	W =  -167.363 deg,	P =     0.000 deg,	R =  -164.964 deg
};
P[653]{
   GP1:
	UF : 7, UT : 3,	CONFIG : 'F U T, 0, 0, 0',
	X =   -22.566  mm,	Y =   363.777  mm,	Z =     0.000  mm,
	W =  -167.363 deg,	P =     0.000 deg,	R =  -161.468 deg
};
P[654]{
   GP1:
	UF : 7, UT : 3,	CONFIG : 'F U T, 0, 0, 0',
	X =   -44.583  mm,	Y =   361.733  mm,	Z =     0.000  mm,
	W =  -167.363 deg,	P =     0.000 deg,	R =  -157.902 deg
};
P[655]{
   GP1:
	UF : 7, UT : 3,	CONFIG : 'F U T, 0, 0, 0',
	X =   -66.134  mm,	Y =   358.425  mm,	Z =     0.000  mm,
	W =  -167.363 deg,	P =     0.000 deg,	R =  -154.243 deg
};
P[656]{
   GP1:
	UF : 7, UT : 3,	CONFIG : 'F U T, 0, 0, 0',
	X =   -66.134  mm,	Y =   358.425  mm,	Z =     0.000  mm,
	W =  -167.363 deg,	P =     0.000 deg,	R =  -154.243 deg
};
P[657]{
   GP1:
	UF : 7, UT : 3,	CONFIG : 'F U T, 0, 0, 0',
	X =   -66.134  mm,	Y =   358.425  mm,	Z =     0.000  mm,
	W =  -167.363 deg,	P =     0.000 deg,	R =  -154.243 deg
};
P[658]{
   GP1:
	UF : 7, UT : 3,	CONFIG : 'F U T, 0, 0, 0',
	X =   -66.134  mm,	Y =   358.425  mm,	Z =     0.000  mm,
	W =  -167.363 deg,	P =     0.000 deg,	R =  -154.243 deg
};
P[659]{
   GP1:
	UF : 7, UT : 3,	CONFIG : 'F U T, 0, 0, 0',
	X =   -95.933  mm,	Y =   351.637  mm,	Z =     0.000  mm,
	W =  -167.364 deg,	P =     0.000 deg,	R =  -149.101 deg
};
P[660]{
   GP1:
	UF : 7, UT : 3,	CONFIG : 'F U T, 0, 0, 0',
	X =   -95.933  mm,	Y =   351.637  mm,	Z =     0.000  mm,
	W =  -167.364 deg,	P =     0.000 deg,	R =  -149.101 deg
};
P[661]{
   GP1:
	UF : 7, UT : 3,	CONFIG : 'F U T, 0, 0, 0',
	X =   -95.933  mm,	Y =   351.637  mm,	Z =     0.000  mm,
	W =  -167.364 deg,	P =     0.000 deg,	R =  -149.101 deg
};
P[662]{
   GP1:
	UF : 7, UT : 3,	CONFIG : 'F U T, 0, 0, 0',
	X =   -95.933  mm,	Y =   351.637  mm,	Z =     0.000  mm,
	W =  -167.364 deg,	P =     0.000 deg,	R =  -149.101 deg
};
P[663]{
   GP1:
	UF : 7, UT : 3,	CONFIG : 'F U T, 0, 0, 0',
	X =  -119.608  mm,	Y =   344.296  mm,	Z =     0.000  mm,
	W =  -167.362 deg,	P =    -0.003 deg,	R =  -145.749 deg
};
P[664]{
   GP1:
	UF : 7, UT : 3,	CONFIG : 'F U T, 0, 0, 0',
	X =  -139.995  mm,	Y =   336.526  mm,	Z =     0.000  mm,
	W =  -167.361 deg,	P =    -0.006 deg,	R =  -142.395 deg
};
P[665]{
   GP1:
	UF : 7, UT : 3,	CONFIG : 'F U T, 0, 0, 0',
	X =  -159.924  mm,	Y =   327.510  mm,	Z =     0.000  mm,
	W =  -167.360 deg,	P =    -0.009 deg,	R =  -139.007 deg
};
P[666]{
   GP1:
	UF : 7, UT : 3,	CONFIG : 'F U T, 0, 0, 0',
	X =  -178.680  mm,	Y =   317.678  mm,	Z =     0.001  mm,
	W =  -167.360 deg,	P =    -0.012 deg,	R =  -135.533 deg
};
P[667]{
   GP1:
	UF : 7, UT : 3,	CONFIG : 'F U T, 0, 0, 0',
	X =  -197.549  mm,	Y =   306.301  mm,	Z =     0.004  mm,
	W =  -167.359 deg,	P =    -0.015 deg,	R =  -132.167 deg
};
P[668]{
   GP1:
	UF : 7, UT : 3,	CONFIG : 'F U T, 0, 0, 0',
	X =  -215.109  mm,	Y =   294.223  mm,	Z =     0.010  mm,
	W =  -167.360 deg,	P =    -0.018 deg,	R =  -128.729 deg
};
P[669]{
   GP1:
	UF : 7, UT : 3,	CONFIG : 'F U T, 0, 0, 0',
	X =  -232.259  mm,	Y =   280.893  mm,	Z =     0.017  mm,
	W =  -167.360 deg,	P =    -0.021 deg,	R =  -125.331 deg
};
P[670]{
   GP1:
	UF : 7, UT : 3,	CONFIG : 'F U T, 0, 0, 0',
	X =  -244.161  mm,	Y =   270.615  mm,	Z =     0.021  mm,
	W =  -167.377 deg,	P =    -0.005 deg,	R =  -122.858 deg
};
P[671]{
   GP1:
	UF : 7, UT : 3,	CONFIG : 'F U T, 0, 0, 0',
	X =  -255.588  mm,	Y =   259.851  mm,	Z =     0.024  mm,
	W =  -167.392 deg,	P =     0.012 deg,	R =  -120.398 deg
};
P[672]{
   GP1:
	UF : 7, UT : 3,	CONFIG : 'F U T, 0, 0, 0',
	X =  -266.547  mm,	Y =   248.605  mm,	Z =     0.021  mm,
	W =  -167.405 deg,	P =     0.031 deg,	R =  -117.928 deg
};
P[673]{
   GP1:
	UF : 7, UT : 3,	CONFIG : 'F U T, 0, 0, 0',
	X =  -276.051  mm,	Y =   238.002  mm,	Z =     0.016  mm,
	W =  -167.466 deg,	P =     0.019 deg,	R =  -115.748 deg
};
P[674]{
   GP1:
	UF : 7, UT : 3,	CONFIG : 'F U T, 0, 0, 0',
	X =  -284.948  mm,	Y =   227.251  mm,	Z =     0.017  mm,
	W =  -167.526 deg,	P =     0.013 deg,	R =  -113.518 deg
};
P[675]{
   GP1:
	UF : 7, UT : 3,	CONFIG : 'F U T, 0, 0, 0',
	X =  -294.786  mm,	Y =   214.339  mm,	Z =     0.044  mm,
	W =  -167.627 deg,	P =    -0.122 deg,	R =  -110.930 deg
};
P[676]{
   GP1:
	UF : 7, UT : 3,	CONFIG : 'F U T, 0, 0, 0',
	X =  -306.175  mm,	Y =   197.743  mm,	Z =     0.197  mm,
	W =  -167.686 deg,	P =    -0.731 deg,	R =  -107.779 deg
};
P[677]{
   GP1:
	UF : 7, UT : 3,	CONFIG : 'F U T, 0, 0, 0',
	X =  -317.263  mm,	Y =   179.431  mm,	Z =     0.730  mm,
	W =  -167.390 deg,	P =    -2.092 deg,	R =  -104.509 deg
};
P[678]{
   GP1:
	UF : 7, UT : 3,	CONFIG : 'F U T, 0, 0, 0',
	X =  -320.981  mm,	Y =   172.696  mm,	Z =     1.000  mm,
	W =  -167.300 deg,	P =    -1.953 deg,	R =  -103.384 deg
};
P[679]{
   GP1:
	UF : 7, UT : 3,	CONFIG : 'F U T, 0, 0, 0',
	X =  -320.981  mm,	Y =   172.696  mm,	Z =     1.000  mm,
	W =  -167.300 deg,	P =    -1.953 deg,	R =  -103.384 deg
};
P[680]{
   GP1:
	UF : 7, UT : 3,	CONFIG : 'F U T, 0, 0, 0',
	X =  -320.981  mm,	Y =   172.696  mm,	Z =     1.000  mm,
	W =  -167.300 deg,	P =    -1.953 deg,	R =  -103.384 deg
};
P[681]{
   GP1:
	UF : 7, UT : 3,	CONFIG : 'F U T, 0, 0, 0',
	X =  -320.981  mm,	Y =   172.696  mm,	Z =     1.000  mm,
	W =  -167.300 deg,	P =    -1.953 deg,	R =  -103.384 deg
};
P[682]{
   GP1:
	UF : 7, UT : 3,	CONFIG : 'F U T, 0, 0, 0',
	X =  -335.149  mm,	Y =   143.280  mm,	Z =     1.000  mm,
	W =  -166.771 deg,	P =     0.958 deg,	R =   -98.400 deg
};
P[683]{
   GP1:
	UF : 7, UT : 3,	CONFIG : 'F U T, 0, 0, 0',
	X =  -335.149  mm,	Y =   143.280  mm,	Z =     1.000  mm,
	W =  -166.771 deg,	P =     0.958 deg,	R =   -98.400 deg
};
P[684]{
   GP1:
	UF : 7, UT : 3,	CONFIG : 'F U T, 0, 0, 0',
	X =  -335.149  mm,	Y =   143.280  mm,	Z =     1.000  mm,
	W =  -166.771 deg,	P =     0.958 deg,	R =   -98.400 deg
};
P[685]{
   GP1:
	UF : 7, UT : 3,	CONFIG : 'F U T, 0, 0, 0',
	X =  -335.149  mm,	Y =   143.280  mm,	Z =     1.000  mm,
	W =  -166.771 deg,	P =     0.958 deg,	R =   -98.400 deg
};
P[686]{
   GP1:
	UF : 7, UT : 3,	CONFIG : 'F U T, 0, 0, 0',
	X =  -339.748  mm,	Y =   131.983  mm,	Z =     0.730  mm,
	W =  -166.786 deg,	P =     1.412 deg,	R =   -96.034 deg
};
P[687]{
   GP1:
	UF : 7, UT : 3,	CONFIG : 'F U T, 0, 0, 0',
	X =  -342.818  mm,	Y =   123.768  mm,	Z =     0.476  mm,
	W =  -167.136 deg,	P =     1.640 deg,	R =   -94.686 deg
};
P[688]{
   GP1:
	UF : 7, UT : 3,	CONFIG : 'F U T, 0, 0, 0',
	X =  -346.796  mm,	Y =   112.170  mm,	Z =     0.189  mm,
	W =  -167.517 deg,	P =     1.060 deg,	R =   -92.897 deg
};
P[689]{
   GP1:
	UF : 7, UT : 3,	CONFIG : 'F U T, 0, 0, 0',
	X =  -351.269  mm,	Y =    97.241  mm,	Z =     0.036  mm,
	W =  -167.527 deg,	P =     0.274 deg,	R =   -90.479 deg
};
P[690]{
   GP1:
	UF : 7, UT : 3,	CONFIG : 'F U T, 0, 0, 0',
	X =  -353.700  mm,	Y =    88.024  mm,	Z =     0.014  mm,
	W =  -167.478 deg,	P =     0.102 deg,	R =   -88.932 deg
};
P[691]{
   GP1:
	UF : 7, UT : 3,	CONFIG : 'F U T, 0, 0, 0',
	X =  -357.903  mm,	Y =    68.887  mm,	Z =     0.006  mm,
	W =  -167.405 deg,	P =     0.015 deg,	R =   -85.835 deg
};
P[692]{
   GP1:
	UF : 7, UT : 3,	CONFIG : 'F U T, 0, 1, 0',
	X =  -361.390  mm,	Y =    47.355  mm,	Z =     0.005  mm,
	W =  -167.391 deg,	P =     0.015 deg,	R =   -82.373 deg
};
P[693]{
   GP1:
	UF : 7, UT : 3,	CONFIG : 'F U T, 0, 1, 0',
	X =  -363.599  mm,	Y =    25.365  mm,	Z =     0.004  mm,
	W =  -167.377 deg,	P =     0.013 deg,	R =   -78.969 deg
};
P[694]{
   GP1:
	UF : 7, UT : 3,	CONFIG : 'F U T, 0, 1, 0',
	X =  -364.492  mm,	Y =     0.000  mm,	Z =     0.000  mm,
	W =  -167.361 deg,	P =     0.009 deg,	R =   -75.580 deg
};
P[695]{
   GP1:
	UF : 7, UT : 3,	CONFIG : 'F U T, 0, 1, 0',
	X =  -364.492  mm,	Y =     0.000  mm,	Z =     0.000  mm,
	W =  -167.361 deg,	P =     0.009 deg,	R =   -75.580 deg
};
P[696]{
   GP1:
	UF : 7, UT : 3,	CONFIG : 'F U T, 0, 1, 0',
	X =  -364.492  mm,	Y =     0.000  mm,	Z =     0.000  mm,
	W =  -167.361 deg,	P =     0.009 deg,	R =   -75.580 deg
};
P[697]{
   GP1:
	UF : 7, UT : 3,	CONFIG : 'F U T, 0, 1, 0',
	X =  -364.492  mm,	Y =     0.000  mm,	Z =     0.000  mm,
	W =  -167.361 deg,	P =     0.009 deg,	R =   -75.580 deg
};
P[698]{
   GP1:
	UF : 7, UT : 3,	CONFIG : 'F U T, 0, 1, 0',
	X =  -361.358  mm,	Y =     0.000  mm,	Z =     0.000  mm,
	W =  -167.361 deg,	P =     0.009 deg,	R =   -75.580 deg
};
P[699]{
   GP1:
	UF : 7, UT : 3,	CONFIG : 'F U T, 0, 1, 0',
	X =  -361.358  mm,	Y =     0.000  mm,	Z =     0.000  mm,
	W =  -167.361 deg,	P =     0.009 deg,	R =   -75.580 deg
};
P[700]{
   GP1:
	UF : 7, UT : 3,	CONFIG : 'F U T, 0, 1, 0',
	X =  -361.358  mm,	Y =     0.000  mm,	Z =     0.000  mm,
	W =  -167.361 deg,	P =     0.009 deg,	R =   -75.580 deg
};
P[701]{
   GP1:
	UF : 7, UT : 3,	CONFIG : 'F U T, 0, 1, 0',
	X =  -361.358  mm,	Y =     0.000  mm,	Z =     0.000  mm,
	W =  -167.361 deg,	P =     0.009 deg,	R =   -75.580 deg
};
P[702]{
   GP1:
	UF : 7, UT : 3,	CONFIG : 'F U T, 0, 1, 0',
	X =  -360.448  mm,	Y =    25.448  mm,	Z =     0.004  mm,
	W =  -167.380 deg,	P =     0.011 deg,	R =   -79.034 deg
};
P[703]{
   GP1:
	UF : 7, UT : 3,	CONFIG : 'F U T, 0, 1, 0',
	X =  -358.205  mm,	Y =    47.576  mm,	Z =     0.004  mm,
	W =  -167.396 deg,	P =     0.011 deg,	R =   -82.501 deg
};
P[704]{
   GP1:
	UF : 7, UT : 3,	CONFIG : 'F U T, 0, 0, 0',
	X =  -354.557  mm,	Y =    69.691  mm,	Z =     0.003  mm,
	W =  -167.412 deg,	P =     0.009 deg,	R =   -85.970 deg
};
P[705]{
   GP1:
	UF : 7, UT : 3,	CONFIG : 'F U T, 0, 0, 0',
	X =  -350.424  mm,	Y =    88.210  mm,	Z =     0.008  mm,
	W =  -167.495 deg,	P =     0.092 deg,	R =   -89.113 deg
};
P[706]{
   GP1:
	UF : 7, UT : 3,	CONFIG : 'F U T, 0, 0, 0',
	X =  -347.970  mm,	Y =    97.380  mm,	Z =     0.026  mm,
	W =  -167.558 deg,	P =     0.268 deg,	R =   -90.637 deg
};
P[707]{
   GP1:
	UF : 7, UT : 3,	CONFIG : 'F U T, 0, 0, 0',
	X =  -343.655  mm,	Y =   111.666  mm,	Z =     0.171  mm,
	W =  -167.608 deg,	P =     1.108 deg,	R =   -93.006 deg
};
P[708]{
   GP1:
	UF : 7, UT : 3,	CONFIG : 'F U T, 0, 0, 0',
	X =  -339.758  mm,	Y =   123.026  mm,	Z =     0.470  mm,
	W =  -167.282 deg,	P =     1.809 deg,	R =   -94.807 deg
};
P[709]{
   GP1:
	UF : 7, UT : 3,	CONFIG : 'F U T, 0, 0, 0',
	X =  -338.361  mm,	Y =   126.823  mm,	Z =     0.600  mm,
	W =  -167.129 deg,	P =     1.834 deg,	R =   -95.529 deg
};
P[710]{
   GP1:
	UF : 7, UT : 3,	CONFIG : 'F U T, 0, 0, 0',
	X =  -334.723  mm,	Y =   136.137  mm,	Z =     0.881  mm,
	W =  -166.917 deg,	P =     1.263 deg,	R =   -97.107 deg
};
P[711]{
   GP1:
	UF : 7, UT : 3,	CONFIG : 'F U T, 0, 0, 0',
	X =  -332.516  mm,	Y =   141.472  mm,	Z =     1.000  mm,
	W =  -166.975 deg,	P =     1.005 deg,	R =   -98.012 deg
};
P[712]{
   GP1:
	UF : 7, UT : 3,	CONFIG : 'F U T, 0, 0, 0',
	X =  -332.516  mm,	Y =   141.472  mm,	Z =     1.000  mm,
	W =  -166.975 deg,	P =     1.005 deg,	R =   -98.012 deg
};
P[713]{
   GP1:
	UF : 7, UT : 3,	CONFIG : 'F U T, 0, 0, 0',
	X =  -332.516  mm,	Y =   141.472  mm,	Z =     1.000  mm,
	W =  -166.975 deg,	P =     1.005 deg,	R =   -98.012 deg
};
P[714]{
   GP1:
	UF : 7, UT : 3,	CONFIG : 'F U T, 0, 0, 0',
	X =  -332.516  mm,	Y =   141.472  mm,	Z =     1.000  mm,
	W =  -166.975 deg,	P =     1.005 deg,	R =   -98.012 deg
};
P[715]{
   GP1:
	UF : 7, UT : 3,	CONFIG : 'F U T, 0, 0, 0',
	X =  -317.920  mm,	Y =   171.762  mm,	Z =     1.000  mm,
	W =  -167.665 deg,	P =    -1.869 deg,	R =  -103.241 deg
};
P[716]{
   GP1:
	UF : 7, UT : 3,	CONFIG : 'F U T, 0, 0, 0',
	X =  -317.920  mm,	Y =   171.762  mm,	Z =     1.000  mm,
	W =  -167.665 deg,	P =    -1.869 deg,	R =  -103.241 deg
};
P[717]{
   GP1:
	UF : 7, UT : 3,	CONFIG : 'F U T, 0, 0, 0',
	X =  -317.920  mm,	Y =   171.762  mm,	Z =     1.000  mm,
	W =  -167.665 deg,	P =    -1.869 deg,	R =  -103.241 deg
};
P[718]{
   GP1:
	UF : 7, UT : 3,	CONFIG : 'F U T, 0, 0, 0',
	X =  -317.920  mm,	Y =   171.762  mm,	Z =     1.000  mm,
	W =  -167.665 deg,	P =    -1.869 deg,	R =  -103.241 deg
};
P[719]{
   GP1:
	UF : 7, UT : 3,	CONFIG : 'F U T, 0, 0, 0',
	X =  -314.044  mm,	Y =   178.741  mm,	Z =     0.714  mm,
	W =  -167.669 deg,	P =    -2.067 deg,	R =  -104.626 deg
};
P[720]{
   GP1:
	UF : 7, UT : 3,	CONFIG : 'F U T, 0, 0, 0',
	X =  -302.748  mm,	Y =   197.275  mm,	Z =     0.167  mm,
	W =  -167.795 deg,	P =    -0.680 deg,	R =  -108.071 deg
};
P[721]{
   GP1:
	UF : 7, UT : 3,	CONFIG : 'F U T, 0, 0, 0',
	X =  -291.275  mm,	Y =   213.833  mm,	Z =     0.025  mm,
	W =  -167.665 deg,	P =    -0.076 deg,	R =  -111.198 deg
};
P[722]{
   GP1:
	UF : 7, UT : 3,	CONFIG : 'F U T, 0, 0, 0',
	X =  -281.263  mm,	Y =   226.842  mm,	Z =     0.007  mm,
	W =  -167.540 deg,	P =     0.044 deg,	R =  -113.765 deg
};
P[723]{
   GP1:
	UF : 7, UT : 3,	CONFIG : 'F U T, 0, 0, 0',
	X =  -272.132  mm,	Y =   237.716  mm,	Z =     0.011  mm,
	W =  -167.474 deg,	P =     0.039 deg,	R =  -116.104 deg
};
P[724]{
   GP1:
	UF : 7, UT : 3,	CONFIG : 'F U T, 0, 0, 0',
	X =  -262.538  mm,	Y =   248.276  mm,	Z =     0.019  mm,
	W =  -167.408 deg,	P =     0.039 deg,	R =  -118.442 deg
};
P[725]{
   GP1:
	UF : 7, UT : 3,	CONFIG : 'F U T, 0, 0, 0',
	X =  -251.581  mm,	Y =   259.374  mm,	Z =     0.023  mm,
	W =  -167.395 deg,	P =     0.018 deg,	R =  -120.883 deg
};
P[726]{
   GP1:
	UF : 7, UT : 3,	CONFIG : 'F U T, 0, 0, 0',
	X =  -240.221  mm,	Y =   269.932  mm,	Z =     0.021  mm,
	W =  -167.380 deg,	P =    -0.002 deg,	R =  -123.334 deg
};
P[727]{
   GP1:
	UF : 7, UT : 3,	CONFIG : 'F U T, 0, 0, 0',
	X =  -228.302  mm,	Y =   280.085  mm,	Z =     0.016  mm,
	W =  -167.364 deg,	P =    -0.020 deg,	R =  -125.793 deg
};
P[728]{
   GP1:
	UF : 7, UT : 3,	CONFIG : 'F U T, 0, 0, 0',
	X =  -211.297  mm,	Y =   293.128  mm,	Z =     0.009  mm,
	W =  -167.363 deg,	P =    -0.018 deg,	R =  -129.084 deg
};
P[729]{
   GP1:
	UF : 7, UT : 3,	CONFIG : 'F U T, 0, 0, 0',
	X =  -194.292  mm,	Y =   304.657  mm,	Z =     0.004  mm,
	W =  -167.362 deg,	P =    -0.015 deg,	R =  -132.493 deg
};
P[730]{
   GP1:
	UF : 7, UT : 3,	CONFIG : 'F U T, 0, 0, 0',
	X =  -176.033  mm,	Y =   315.568  mm,	Z =     0.001  mm,
	W =  -167.362 deg,	P =    -0.012 deg,	R =  -135.789 deg
};
P[731]{
   GP1:
	UF : 7, UT : 3,	CONFIG : 'F U T, 0, 0, 0',
	X =  -157.288  mm,	Y =   325.309  mm,	Z =     0.000  mm,
	W =  -167.362 deg,	P =    -0.009 deg,	R =  -139.100 deg
};
P[732]{
   GP1:
	UF : 7, UT : 3,	CONFIG : 'F U T, 0, 0, 0',
	X =  -138.454  mm,	Y =   333.763  mm,	Z =     0.000  mm,
	W =  -167.362 deg,	P =    -0.006 deg,	R =  -142.478 deg
};
P[733]{
   GP1:
	UF : 7, UT : 3,	CONFIG : 'F U T, 0, 0, 0',
	X =  -118.401  mm,	Y =   341.400  mm,	Z =     0.000  mm,
	W =  -167.363 deg,	P =    -0.003 deg,	R =  -145.771 deg
};
P[734]{
   GP1:
	UF : 7, UT : 3,	CONFIG : 'F U T, 0, 0, 0',
	X =   -95.742  mm,	Y =   348.434  mm,	Z =     0.000  mm,
	W =  -167.364 deg,	P =     0.000 deg,	R =  -149.103 deg
};
P[735]{
   GP1:
	UF : 7, UT : 3,	CONFIG : 'F U T, 0, 0, 0',
	X =   -95.742  mm,	Y =   348.434  mm,	Z =     0.000  mm,
	W =  -167.364 deg,	P =     0.000 deg,	R =  -149.103 deg
};
P[736]{
   GP1:
	UF : 7, UT : 3,	CONFIG : 'F U T, 0, 0, 0',
	X =   -95.742  mm,	Y =   348.434  mm,	Z =     0.000  mm,
	W =  -167.364 deg,	P =     0.000 deg,	R =  -149.103 deg
};
P[737]{
   GP1:
	UF : 7, UT : 3,	CONFIG : 'F U T, 0, 0, 0',
	X =   -95.742  mm,	Y =   348.434  mm,	Z =     0.000  mm,
	W =  -167.364 deg,	P =     0.000 deg,	R =  -149.103 deg
};
P[738]{
   GP1:
	UF : 7, UT : 3,	CONFIG : 'F U T, 0, 0, 0',
	X =   -64.916  mm,	Y =   355.467  mm,	Z =     0.000  mm,
	W =  -167.363 deg,	P =     0.000 deg,	R =  -154.628 deg
};
P[739]{
   GP1:
	UF : 7, UT : 3,	CONFIG : 'F U T, 0, 0, 0',
	X =   -64.916  mm,	Y =   355.467  mm,	Z =     0.000  mm,
	W =  -167.363 deg,	P =     0.000 deg,	R =  -154.628 deg
};
P[740]{
   GP1:
	UF : 7, UT : 3,	CONFIG : 'F U T, 0, 0, 0',
	X =   -64.916  mm,	Y =   355.467  mm,	Z =     0.000  mm,
	W =  -167.363 deg,	P =     0.000 deg,	R =  -154.628 deg
};
P[741]{
   GP1:
	UF : 7, UT : 3,	CONFIG : 'F U T, 0, 0, 0',
	X =   -64.916  mm,	Y =   355.467  mm,	Z =     0.000  mm,
	W =  -167.363 deg,	P =     0.000 deg,	R =  -154.628 deg
};
P[742]{
   GP1:
	UF : 7, UT : 3,	CONFIG : 'F U T, 0, 0, 0',
	X =   -43.097  mm,	Y =   358.757  mm,	Z =     0.000  mm,
	W =  -167.363 deg,	P =     0.000 deg,	R =  -158.018 deg
};
P[743]{
   GP1:
	UF : 7, UT : 3,	CONFIG : 'F U T, 0, 0, 0',
	X =   -21.980  mm,	Y =   360.671  mm,	Z =     0.000  mm,
	W =  -167.363 deg,	P =     0.000 deg,	R =  -161.549 deg
};
P[744]{
   GP1:
	UF : 7, UT : 3,	CONFIG : 'F U T, 0, 0, 0',
	X =     0.061  mm,	Y =   361.358  mm,	Z =     0.000  mm,
	W =  -167.363 deg,	P =     0.000 deg,	R =  -164.959 deg
};
P[745]{
   GP1:
	UF : 7, UT : 3,	CONFIG : 'F U T, 0, 0, 0',
	X =    22.208  mm,	Y =   360.659  mm,	Z =     0.000  mm,
	W =  -167.363 deg,	P =     0.000 deg,	R =  -168.353 deg
};
P[746]{
   GP1:
	UF : 7, UT : 3,	CONFIG : 'F U T, 0, 0, 0',
	X =    43.255  mm,	Y =   358.738  mm,	Z =     0.000  mm,
	W =  -167.363 deg,	P =     0.000 deg,	R =  -171.883 deg
};
P[747]{
   GP1:
	UF : 7, UT : 3,	CONFIG : 'F U T, 0, 0, 0',
	X =    64.916  mm,	Y =   355.467  mm,	Z =     0.000  mm,
	W =  -167.363 deg,	P =     0.000 deg,	R =  -175.272 deg
};
P[748]{
   GP1:
	UF : 7, UT : 3,	CONFIG : 'F U T, 0, 0, 0',
	X =    64.916  mm,	Y =   355.467  mm,	Z =     0.000  mm,
	W =  -167.363 deg,	P =     0.000 deg,	R =  -175.272 deg
};
P[749]{
   GP1:
	UF : 7, UT : 3,	CONFIG : 'F U T, 0, 0, 0',
	X =    64.916  mm,	Y =   355.467  mm,	Z =     0.000  mm,
	W =  -167.363 deg,	P =     0.000 deg,	R =  -175.272 deg
};
P[750]{
   GP1:
	UF : 7, UT : 3,	CONFIG : 'F U T, 0, 0, 0',
	X =    64.916  mm,	Y =   355.467  mm,	Z =     0.000  mm,
	W =  -167.363 deg,	P =     0.000 deg,	R =  -175.272 deg
};
P[751]{
   GP1:
	UF : 7, UT : 3,	CONFIG : 'F U T, 0, 0, 0',
	X =    95.742  mm,	Y =   348.434  mm,	Z =     0.000  mm,
	W =  -167.363 deg,	P =     0.000 deg,	R =   179.209 deg
};
P[752]{
   GP1:
	UF : 7, UT : 3,	CONFIG : 'F U T, 0, 0, 0',
	X =    95.742  mm,	Y =   348.434  mm,	Z =     0.000  mm,
	W =  -167.363 deg,	P =     0.000 deg,	R =   179.209 deg
};
P[753]{
   GP1:
	UF : 7, UT : 3,	CONFIG : 'F U T, 0, 0, 0',
	X =    95.742  mm,	Y =   348.434  mm,	Z =     0.000  mm,
	W =  -167.363 deg,	P =     0.000 deg,	R =   179.209 deg
};
P[754]{
   GP1:
	UF : 7, UT : 3,	CONFIG : 'F U T, 0, 0, 0',
	X =    95.742  mm,	Y =   348.434  mm,	Z =     0.000  mm,
	W =  -167.363 deg,	P =     0.000 deg,	R =   179.209 deg
};
P[755]{
   GP1:
	UF : 7, UT : 3,	CONFIG : 'F U T, 0, 0, 0',
	X =   121.471  mm,	Y =   340.308  mm,	Z =     0.000  mm,
	W =  -167.363 deg,	P =     0.000 deg,	R =   175.407 deg
};
P[756]{
   GP1:
	UF : 7, UT : 3,	CONFIG : 'F U T, 0, 0, 0',
	X =   143.916  mm,	Y =   331.439  mm,	Z =     0.000  mm,
	W =  -167.364 deg,	P =     0.000 deg,	R =   171.611 deg
};
P[757]{
   GP1:
	UF : 7, UT : 3,	CONFIG : 'F U T, 0, 0, 0',
	X =   165.675  mm,	Y =   321.118  mm,	Z =     0.000  mm,
	W =  -167.364 deg,	P =     0.000 deg,	R =   167.801 deg
};
P[758]{
   GP1:
	UF : 7, UT : 3,	CONFIG : 'F U T, 0, 0, 0',
	X =   186.459  mm,	Y =   309.511  mm,	Z =     0.000  mm,
	W =  -167.364 deg,	P =     0.000 deg,	R =   163.968 deg
};
P[759]{
   GP1:
	UF : 7, UT : 3,	CONFIG : 'F U T, 0, 0, 0',
	X =   206.624  mm,	Y =   296.430  mm,	Z =     0.000  mm,
	W =  -167.364 deg,	P =     0.000 deg,	R =   160.166 deg
};
P[760]{
   GP1:
	UF : 7, UT : 3,	CONFIG : 'F U T, 0, 0, 0',
	X =   225.736  mm,	Y =   282.147  mm,	Z =     0.000  mm,
	W =  -167.364 deg,	P =     0.000 deg,	R =   156.350 deg
};
P[761]{
   GP1:
	UF : 7, UT : 3,	CONFIG : 'F U T, 0, 0, 0',
	X =   244.345  mm,	Y =   266.195  mm,	Z =     0.000  mm,
	W =  -167.364 deg,	P =     0.000 deg,	R =   152.581 deg
};
P[762]{
   GP1:
	UF : 7, UT : 3,	CONFIG : 'F U T, 0, 0, 0',
	X =   261.258  mm,	Y =   249.618  mm,	Z =     0.000  mm,
	W =  -167.364 deg,	P =     0.000 deg,	R =   148.718 deg
};
P[763]{
   GP1:
	UF : 7, UT : 3,	CONFIG : 'F U T, 0, 0, 0',
	X =   277.507  mm,	Y =   231.417  mm,	Z =     0.000  mm,
	W =  -167.364 deg,	P =     0.000 deg,	R =   144.979 deg
};
P[764]{
   GP1:
	UF : 7, UT : 3,	CONFIG : 'F U T, 0, 0, 0',
	X =   292.091  mm,	Y =   212.720  mm,	Z =     0.000  mm,
	W =  -167.364 deg,	P =     0.000 deg,	R =   141.122 deg
};
P[765]{
   GP1:
	UF : 7, UT : 3,	CONFIG : 'F U T, 0, 0, 0',
	X =   305.767  mm,	Y =   192.539  mm,	Z =     0.000  mm,
	W =  -167.364 deg,	P =     0.000 deg,	R =   137.342 deg
};
P[766]{
   GP1:
	UF : 7, UT : 3,	CONFIG : 'F U T, 0, 0, 0',
	X =   318.385  mm,	Y =   170.874  mm,	Z =     0.000  mm,
	W =  -167.364 deg,	P =     0.000 deg,	R =   133.523 deg
};
P[767]{
   GP1:
	UF : 7, UT : 3,	CONFIG : 'F U T, 0, 0, 0',
	X =   318.385  mm,	Y =   170.874  mm,	Z =     0.000  mm,
	W =  -167.364 deg,	P =     0.000 deg,	R =   133.523 deg
};
P[768]{
   GP1:
	UF : 7, UT : 3,	CONFIG : 'F U T, 0, 0, 0',
	X =   318.385  mm,	Y =   170.874  mm,	Z =     0.000  mm,
	W =  -167.364 deg,	P =     0.000 deg,	R =   133.523 deg
};
P[769]{
   GP1:
	UF : 7, UT : 3,	CONFIG : 'F U T, 0, 0, 0',
	X =   318.385  mm,	Y =   170.874  mm,	Z =     0.000  mm,
	W =  -167.364 deg,	P =     0.000 deg,	R =   133.523 deg
};
P[770]{
   GP1:
	UF : 7, UT : 3,	CONFIG : 'F U T, 0, 0, 0',
	X =   332.104  mm,	Y =   142.381  mm,	Z =     0.000  mm,
	W =  -167.363 deg,	P =     0.001 deg,	R =   128.768 deg
};
P[771]{
   GP1:
	UF : 7, UT : 3,	CONFIG : 'F U T, 0, 0, 0',
	X =   332.104  mm,	Y =   142.381  mm,	Z =     0.000  mm,
	W =  -167.363 deg,	P =     0.001 deg,	R =   128.768 deg
};
P[772]{
   GP1:
	UF : 7, UT : 3,	CONFIG : 'F U T, 0, 0, 0',
	X =   332.104  mm,	Y =   142.381  mm,	Z =     0.000  mm,
	W =  -167.363 deg,	P =     0.001 deg,	R =   128.768 deg
};
P[773]{
   GP1:
	UF : 7, UT : 3,	CONFIG : 'F U T, 0, 0, 0',
	X =   332.104  mm,	Y =   142.381  mm,	Z =     0.000  mm,
	W =  -167.363 deg,	P =     0.001 deg,	R =   128.768 deg
};
P[774]{
   GP1:
	UF : 7, UT : 3,	CONFIG : 'F U T, 0, 0, 0',
	X =   340.331  mm,	Y =   121.401  mm,	Z =     0.000  mm,
	W =  -167.363 deg,	P =     0.000 deg,	R =   124.654 deg
};
P[775]{
   GP1:
	UF : 7, UT : 3,	CONFIG : 'F U T, 0, 0, 0',
	X =   347.718  mm,	Y =    98.269  mm,	Z =     0.000  mm,
	W =  -167.364 deg,	P =     0.000 deg,	R =   120.888 deg
};
P[776]{
   GP1:
	UF : 7, UT : 3,	CONFIG : 'F U T, 0, 0, 0',
	X =   353.411  mm,	Y =    75.263  mm,	Z =     0.000  mm,
	W =  -167.364 deg,	P =     0.000 deg,	R =   117.027 deg
};
P[777]{
   GP1:
	UF : 7, UT : 3,	CONFIG : 'F U T, 0, 0, 0',
	X =   357.697  mm,	Y =    51.157  mm,	Z =     0.000  mm,
	W =  -167.364 deg,	P =     0.000 deg,	R =   113.281 deg
};
P[778]{
   GP1:
	UF : 7, UT : 3,	CONFIG : 'F U T, 0, 0, 0',
	X =   360.272  mm,	Y =    27.720  mm,	Z =     0.000  mm,
	W =  -167.364 deg,	P =     0.000 deg,	R =   109.419 deg
};
P[779]{
   GP1:
	UF : 7, UT : 3,	CONFIG : 'F U T, 0, 0, 0',
	X =   361.358  mm,	Y =     0.000  mm,	Z =     0.000  mm,
	W =  -167.364 deg,	P =    -0.001 deg,	R =   105.687 deg
};
P[780]{
   GP1:
	UF : 7, UT : 3,	CONFIG : 'F U T, 0, 0, 0',
	X =   361.358  mm,	Y =     0.000  mm,	Z =     0.000  mm,
	W =  -167.364 deg,	P =    -0.001 deg,	R =   105.687 deg
};
P[781]{
   GP1:
	UF : 7, UT : 3,	CONFIG : 'F U T, 0, 0, 0',
	X =   361.358  mm,	Y =     0.000  mm,	Z =     0.000  mm,
	W =  -167.364 deg,	P =    -0.001 deg,	R =   105.687 deg
};
P[782]{
   GP1:
	UF : 7, UT : 3,	CONFIG : 'F U T, 0, 0, 0',
	X =   361.358  mm,	Y =     0.000  mm,	Z =     0.000  mm,
	W =  -167.364 deg,	P =    -0.001 deg,	R =   105.687 deg
};
P[783]{
   GP1:
	UF : 7, UT : 3,	CONFIG : 'F U T, 0, 0, 0',
	X =   358.223  mm,	Y =     0.000  mm,	Z =     0.000  mm,
	W =  -167.364 deg,	P =    -0.001 deg,	R =   105.690 deg
};
P[784]{
   GP1:
	UF : 7, UT : 3,	CONFIG : 'F U T, 0, 0, 0',
	X =   358.223  mm,	Y =     0.000  mm,	Z =     0.000  mm,
	W =  -167.364 deg,	P =    -0.001 deg,	R =   105.690 deg
};
P[785]{
   GP1:
	UF : 7, UT : 3,	CONFIG : 'F U T, 0, 0, 0',
	X =   358.223  mm,	Y =     0.000  mm,	Z =     0.000  mm,
	W =  -167.364 deg,	P =    -0.001 deg,	R =   105.690 deg
};
P[786]{
   GP1:
	UF : 7, UT : 3,	CONFIG : 'F U T, 0, 0, 0',
	X =   358.223  mm,	Y =     0.000  mm,	Z =     0.000  mm,
	W =  -167.364 deg,	P =    -0.001 deg,	R =   105.690 deg
};
P[787]{
   GP1:
	UF : 7, UT : 3,	CONFIG : 'F U T, 0, 0, 0',
	X =   357.363  mm,	Y =    24.688  mm,	Z =     0.000  mm,
	W =  -167.364 deg,	P =     0.000 deg,	R =   109.041 deg
};
P[788]{
   GP1:
	UF : 7, UT : 3,	CONFIG : 'F U T, 0, 0, 0',
	X =   355.202  mm,	Y =    46.357  mm,	Z =     0.000  mm,
	W =  -167.364 deg,	P =     0.000 deg,	R =   112.450 deg
};
P[789]{
   GP1:
	UF : 7, UT : 3,	CONFIG : 'F U T, 0, 0, 0',
	X =   351.158  mm,	Y =    70.794  mm,	Z =     0.000  mm,
	W =  -167.364 deg,	P =     0.001 deg,	R =   115.826 deg
};
P[790]{
   GP1:
	UF : 7, UT : 3,	CONFIG : 'F U T, 0, 0, 0',
	X =   351.158  mm,	Y =    70.794  mm,	Z =     0.000  mm,
	W =  -167.364 deg,	P =     0.001 deg,	R =   115.826 deg
};
P[791]{
   GP1:
	UF : 7, UT : 3,	CONFIG : 'F U T, 0, 0, 0',
	X =   351.158  mm,	Y =    70.794  mm,	Z =     0.000  mm,
	W =  -167.364 deg,	P =     0.001 deg,	R =   115.826 deg
};
P[792]{
   GP1:
	UF : 7, UT : 3,	CONFIG : 'F U T, 0, 0, 0',
	X =   351.158  mm,	Y =    70.794  mm,	Z =     0.000  mm,
	W =  -167.364 deg,	P =     0.001 deg,	R =   115.826 deg
};
P[793]{
   GP1:
	UF : 7, UT : 3,	CONFIG : 'F U T, 0, 0, 0',
	X =   347.068  mm,	Y =    88.627  mm,	Z =     0.000  mm,
	W =  -167.365 deg,	P =     0.000 deg,	R =   119.442 deg
};
P[794]{
   GP1:
	UF : 7, UT : 3,	CONFIG : 'F U T, 0, 0, 0',
	X =   347.068  mm,	Y =    88.627  mm,	Z =     0.000  mm,
	W =  -167.365 deg,	P =     0.000 deg,	R =   119.442 deg
};
P[795]{
   GP1:
	UF : 7, UT : 3,	CONFIG : 'F U T, 0, 0, 0',
	X =   347.068  mm,	Y =    88.627  mm,	Z =     0.000  mm,
	W =  -167.365 deg,	P =     0.000 deg,	R =   119.442 deg
};
P[796]{
   GP1:
	UF : 7, UT : 3,	CONFIG : 'F U T, 0, 0, 0',
	X =   347.068  mm,	Y =    88.627  mm,	Z =     0.000  mm,
	W =  -167.365 deg,	P =     0.000 deg,	R =   119.442 deg
};
P[797]{
   GP1:
	UF : 7, UT : 3,	CONFIG : 'F U T, 0, 0, 0',
	X =   341.771  mm,	Y =   107.262  mm,	Z =     0.000  mm,
	W =  -167.364 deg,	P =     0.000 deg,	R =   122.386 deg
};
P[798]{
   GP1:
	UF : 7, UT : 3,	CONFIG : 'F U T, 0, 0, 0',
	X =   335.780  mm,	Y =   124.783  mm,	Z =     0.000  mm,
	W =  -167.364 deg,	P =     0.000 deg,	R =   125.464 deg
};
P[799]{
   GP1:
	UF : 7, UT : 3,	CONFIG : 'F U T, 0, 0, 0',
	X =   329.229  mm,	Y =   141.133  mm,	Z =     0.000  mm,
	W =  -167.363 deg,	P =     0.001 deg,	R =   128.775 deg
};
P[800]{
   GP1:
	UF : 7, UT : 3,	CONFIG : 'F U T, 0, 0, 0',
	X =   329.229  mm,	Y =   141.133  mm,	Z =     0.000  mm,
	W =  -167.363 deg,	P =     0.001 deg,	R =   128.775 deg
};
P[801]{
   GP1:
	UF : 7, UT : 3,	CONFIG : 'F U T, 0, 0, 0',
	X =   329.229  mm,	Y =   141.133  mm,	Z =     0.000  mm,
	W =  -167.363 deg,	P =     0.001 deg,	R =   128.775 deg
};
P[802]{
   GP1:
	UF : 7, UT : 3,	CONFIG : 'F U T, 0, 0, 0',
	X =   329.229  mm,	Y =   141.133  mm,	Z =     0.000  mm,
	W =  -167.363 deg,	P =     0.001 deg,	R =   128.775 deg
};
P[803]{
   GP1:
	UF : 7, UT : 3,	CONFIG : 'F U T, 0, 0, 0',
	X =   315.614  mm,	Y =   169.408  mm,	Z =     0.000  mm,
	W =  -167.364 deg,	P =     0.000 deg,	R =   133.481 deg
};
P[804]{
   GP1:
	UF : 7, UT : 3,	CONFIG : 'F U T, 0, 0, 0',
	X =   315.614  mm,	Y =   169.408  mm,	Z =     0.000  mm,
	W =  -167.364 deg,	P =     0.000 deg,	R =   133.481 deg
};
P[805]{
   GP1:
	UF : 7, UT : 3,	CONFIG : 'F U T, 0, 0, 0',
	X =   315.614  mm,	Y =   169.408  mm,	Z =     0.000  mm,
	W =  -167.364 deg,	P =     0.000 deg,	R =   133.481 deg
};
P[806]{
   GP1:
	UF : 7, UT : 3,	CONFIG : 'F U T, 0, 0, 0',
	X =   315.614  mm,	Y =   169.408  mm,	Z =     0.000  mm,
	W =  -167.364 deg,	P =     0.000 deg,	R =   133.481 deg
};
P[807]{
   GP1:
	UF : 7, UT : 3,	CONFIG : 'F U T, 0, 0, 0',
	X =   305.903  mm,	Y =   186.375  mm,	Z =     0.000  mm,
	W =  -167.364 deg,	P =     0.000 deg,	R =   136.350 deg
};
P[808]{
   GP1:
	UF : 7, UT : 3,	CONFIG : 'F U T, 0, 0, 0',
	X =   295.980  mm,	Y =   201.772  mm,	Z =     0.000  mm,
	W =  -167.364 deg,	P =     0.000 deg,	R =   139.338 deg
};
P[809]{
   GP1:
	UF : 7, UT : 3,	CONFIG : 'F U T, 0, 0, 0',
	X =   285.683  mm,	Y =   216.095  mm,	Z =     0.000  mm,
	W =  -167.365 deg,	P =     0.001 deg,	R =   142.509 deg
};
P[810]{
   GP1:
	UF : 7, UT : 3,	CONFIG : 'F U T, 0, 0, 0',
	X =   285.683  mm,	Y =   216.095  mm,	Z =     0.000  mm,
	W =  -167.365 deg,	P =     0.001 deg,	R =   142.509 deg
};
P[811]{
   GP1:
	UF : 7, UT : 3,	CONFIG : 'F U T, 0, 0, 0',
	X =   285.683  mm,	Y =   216.095  mm,	Z =     0.000  mm,
	W =  -167.365 deg,	P =     0.001 deg,	R =   142.509 deg
};
P[812]{
   GP1:
	UF : 7, UT : 3,	CONFIG : 'F U T, 0, 0, 0',
	X =   285.683  mm,	Y =   216.095  mm,	Z =     0.000  mm,
	W =  -167.365 deg,	P =     0.001 deg,	R =   142.509 deg
};
P[813]{
   GP1:
	UF : 7, UT : 3,	CONFIG : 'F U T, 0, 0, 0',
	X =   274.234  mm,	Y =   230.444  mm,	Z =     0.000  mm,
	W =  -167.365 deg,	P =     0.000 deg,	R =   144.557 deg
};
P[814]{
   GP1:
	UF : 7, UT : 3,	CONFIG : 'F U T, 0, 0, 0',
	X =   274.234  mm,	Y =   230.444  mm,	Z =     0.000  mm,
	W =  -167.365 deg,	P =     0.000 deg,	R =   144.557 deg
};
P[815]{
   GP1:
	UF : 7, UT : 3,	CONFIG : 'F U T, 0, 0, 0',
	X =   274.234  mm,	Y =   230.444  mm,	Z =     0.000  mm,
	W =  -167.365 deg,	P =     0.000 deg,	R =   144.557 deg
};
P[816]{
   GP1:
	UF : 7, UT : 3,	CONFIG : 'F U T, 0, 0, 0',
	X =   274.234  mm,	Y =   230.444  mm,	Z =     0.000  mm,
	W =  -167.365 deg,	P =     0.000 deg,	R =   144.557 deg
};
P[817]{
   GP1:
	UF : 7, UT : 3,	CONFIG : 'F U T, 0, 0, 0',
	X =   259.173  mm,	Y =   247.263  mm,	Z =     0.000  mm,
	W =  -167.365 deg,	P =     0.000 deg,	R =   148.734 deg
};
P[818]{
   GP1:
	UF : 7, UT : 3,	CONFIG : 'F U T, 0, 0, 0',
	X =   241.882  mm,	Y =   264.201  mm,	Z =     0.000  mm,
	W =  -167.364 deg,	P =     0.000 deg,	R =   152.581 deg
};
P[819]{
   GP1:
	UF : 7, UT : 3,	CONFIG : 'F U T, 0, 0, 0',
	X =   223.379  mm,	Y =   280.019  mm,	Z =     0.000  mm,
	W =  -167.364 deg,	P =     0.000 deg,	R =   156.446 deg
};
P[820]{
   GP1:
	UF : 7, UT : 3,	CONFIG : 'F U T, 0, 0, 0',
	X =   203.978  mm,	Y =   294.454  mm,	Z =     0.000  mm,
	W =  -167.364 deg,	P =     0.000 deg,	R =   160.281 deg
};
P[821]{
   GP1:
	UF : 7, UT : 3,	CONFIG : 'F U T, 0, 0, 0',
	X =   183.850  mm,	Y =   307.427  mm,	Z =     0.000  mm,
	W =  -167.364 deg,	P =     0.000 deg,	R =   164.143 deg
};
P[822]{
   GP1:
	UF : 7, UT : 3,	CONFIG : 'F U T, 0, 0, 0',
	X =   163.645  mm,	Y =   318.636  mm,	Z =     0.000  mm,
	W =  -167.364 deg,	P =     0.000 deg,	R =   168.167 deg
};
P[823]{
   GP1:
	UF : 7, UT : 3,	CONFIG : 'F U T, 0, 0, 0',
	X =   163.645  mm,	Y =   318.636  mm,	Z =     0.000  mm,
	W =  -167.364 deg,	P =     0.000 deg,	R =   168.167 deg
};
P[824]{
   GP1:
	UF : 7, UT : 3,	CONFIG : 'F U T, 0, 0, 0',
	X =   163.645  mm,	Y =   318.636  mm,	Z =     0.000  mm,
	W =  -167.364 deg,	P =     0.000 deg,	R =   168.167 deg
};
P[825]{
   GP1:
	UF : 7, UT : 3,	CONFIG : 'F U T, 0, 0, 0',
	X =   163.645  mm,	Y =   318.636  mm,	Z =     0.000  mm,
	W =  -167.364 deg,	P =     0.000 deg,	R =   168.167 deg
};
P[826]{
   GP1:
	UF : 7, UT : 3,	CONFIG : 'F U T, 0, 0, 0',
	X =   147.137  mm,	Y =   326.600  mm,	Z =     0.000  mm,
	W =  -167.364 deg,	P =     0.000 deg,	R =   170.957 deg
};
P[827]{
   GP1:
	UF : 7, UT : 3,	CONFIG : 'F U T, 0, 0, 0',
	X =   147.137  mm,	Y =   326.600  mm,	Z =     0.000  mm,
	W =  -167.364 deg,	P =     0.000 deg,	R =   170.957 deg
};
P[828]{
   GP1:
	UF : 7, UT : 3,	CONFIG : 'F U T, 0, 0, 0',
	X =   147.137  mm,	Y =   326.600  mm,	Z =     0.000  mm,
	W =  -167.364 deg,	P =     0.000 deg,	R =   170.957 deg
};
P[829]{
   GP1:
	UF : 7, UT : 3,	CONFIG : 'F U T, 0, 0, 0',
	X =   147.137  mm,	Y =   326.600  mm,	Z =     0.000  mm,
	W =  -167.364 deg,	P =     0.000 deg,	R =   170.957 deg
};
P[830]{
   GP1:
	UF : 7, UT : 3,	CONFIG : 'F U T, 0, 0, 0',
	X =   130.576  mm,	Y =   333.563  mm,	Z =     0.000  mm,
	W =  -167.364 deg,	P =     0.000 deg,	R =   173.741 deg
};
P[831]{
   GP1:
	UF : 7, UT : 3,	CONFIG : 'F U T, 0, 0, 0',
	X =   113.610  mm,	Y =   339.710  mm,	Z =     0.000  mm,
	W =  -167.364 deg,	P =     0.000 deg,	R =   176.553 deg
};
P[832]{
   GP1:
	UF : 7, UT : 3,	CONFIG : 'F U T, 0, 0, 0',
	X =    94.934  mm,	Y =   345.405  mm,	Z =     0.000  mm,
	W =  -167.363 deg,	P =     0.000 deg,	R =   179.177 deg
};
P[833]{
   GP1:
	UF : 7, UT : 3,	CONFIG : 'F U T, 0, 0, 0',
	X =    94.934  mm,	Y =   345.405  mm,	Z =     0.000  mm,
	W =  -167.363 deg,	P =     0.000 deg,	R =   179.177 deg
};
P[834]{
   GP1:
	UF : 7, UT : 3,	CONFIG : 'F U T, 0, 0, 0',
	X =    94.934  mm,	Y =   345.405  mm,	Z =     0.000  mm,
	W =  -167.363 deg,	P =     0.000 deg,	R =   179.177 deg
};
P[835]{
   GP1:
	UF : 7, UT : 3,	CONFIG : 'F U T, 0, 0, 0',
	X =    94.934  mm,	Y =   345.405  mm,	Z =     0.000  mm,
	W =  -167.363 deg,	P =     0.000 deg,	R =   179.177 deg
};
P[836]{
   GP1:
	UF : 7, UT : 3,	CONFIG : 'F U T, 0, 0, 0',
	X =    64.334  mm,	Y =   352.387  mm,	Z =     0.000  mm,
	W =  -167.363 deg,	P =     0.000 deg,	R =  -175.257 deg
};
P[837]{
   GP1:
	UF : 7, UT : 3,	CONFIG : 'F U T, 0, 0, 0',
	X =    64.334  mm,	Y =   352.387  mm,	Z =     0.000  mm,
	W =  -167.363 deg,	P =     0.000 deg,	R =  -175.257 deg
};
P[838]{
   GP1:
	UF : 7, UT : 3,	CONFIG : 'F U T, 0, 0, 0',
	X =    64.334  mm,	Y =   352.387  mm,	Z =     0.000  mm,
	W =  -167.363 deg,	P =     0.000 deg,	R =  -175.257 deg
};
P[839]{
   GP1:
	UF : 7, UT : 3,	CONFIG : 'F U T, 0, 0, 0',
	X =    64.334  mm,	Y =   352.387  mm,	Z =     0.000  mm,
	W =  -167.363 deg,	P =     0.000 deg,	R =  -175.257 deg
};
P[840]{
   GP1:
	UF : 7, UT : 3,	CONFIG : 'F U T, 0, 0, 0',
	X =    46.727  mm,	Y =   355.150  mm,	Z =     0.000  mm,
	W =  -167.363 deg,	P =     0.000 deg,	R =  -172.411 deg
};
P[841]{
   GP1:
	UF : 7, UT : 3,	CONFIG : 'F U T, 0, 0, 0',
	X =    28.906  mm,	Y =   357.038  mm,	Z =     0.000  mm,
	W =  -167.363 deg,	P =     0.000 deg,	R =  -169.566 deg
};
P[842]{
   GP1:
	UF : 7, UT : 3,	CONFIG : 'F U T, 0, 0, 0',
	X =     9.146  mm,	Y =   358.095  mm,	Z =     0.000  mm,
	W =  -167.364 deg,	P =     0.000 deg,	R =  -166.872 deg
};
P[843]{
   GP1:
	UF : 7, UT : 3,	CONFIG : 'F U T, 0, 0, 0',
	X =     9.146  mm,	Y =   358.095  mm,	Z =     0.000  mm,
	W =  -167.364 deg,	P =     0.000 deg,	R =  -166.872 deg
};
P[844]{
   GP1:
	UF : 7, UT : 3,	CONFIG : 'F U T, 0, 0, 0',
	X =     9.146  mm,	Y =   358.095  mm,	Z =     0.000  mm,
	W =  -167.364 deg,	P =     0.000 deg,	R =  -166.872 deg
};
P[845]{
   GP1:
	UF : 7, UT : 3,	CONFIG : 'F U T, 0, 0, 0',
	X =     9.146  mm,	Y =   358.095  mm,	Z =     0.000  mm,
	W =  -167.364 deg,	P =     0.000 deg,	R =  -166.872 deg
};
P[846]{
   GP1:
	UF : 7, UT : 3,	CONFIG : 'F U T, 0, 0, 0',
	X =    -9.146  mm,	Y =   358.095  mm,	Z =     0.000  mm,
	W =  -167.364 deg,	P =     0.000 deg,	R =  -163.020 deg
};
P[847]{
   GP1:
	UF : 7, UT : 3,	CONFIG : 'F U T, 0, 0, 0',
	X =    -9.146  mm,	Y =   358.095  mm,	Z =     0.000  mm,
	W =  -167.364 deg,	P =     0.000 deg,	R =  -163.020 deg
};
P[848]{
   GP1:
	UF : 7, UT : 3,	CONFIG : 'F U T, 0, 0, 0',
	X =    -9.146  mm,	Y =   358.095  mm,	Z =     0.000  mm,
	W =  -167.364 deg,	P =     0.000 deg,	R =  -163.020 deg
};
P[849]{
   GP1:
	UF : 7, UT : 3,	CONFIG : 'F U T, 0, 0, 0',
	X =    -9.146  mm,	Y =   358.095  mm,	Z =     0.000  mm,
	W =  -167.364 deg,	P =     0.000 deg,	R =  -163.020 deg
};
P[850]{
   GP1:
	UF : 7, UT : 3,	CONFIG : 'F U T, 0, 0, 0',
	X =   -28.876  mm,	Y =   357.041  mm,	Z =     0.000  mm,
	W =  -167.364 deg,	P =     0.000 deg,	R =  -160.353 deg
};
P[851]{
   GP1:
	UF : 7, UT : 3,	CONFIG : 'F U T, 0, 0, 0',
	X =   -46.635  mm,	Y =   355.162  mm,	Z =     0.000  mm,
	W =  -167.363 deg,	P =     0.000 deg,	R =  -157.502 deg
};
P[852]{
   GP1:
	UF : 7, UT : 3,	CONFIG : 'F U T, 0, 0, 0',
	X =   -64.334  mm,	Y =   352.387  mm,	Z =     0.000  mm,
	W =  -167.363 deg,	P =     0.000 deg,	R =  -154.648 deg
};
P[853]{
   GP1:
	UF : 7, UT : 3,	CONFIG : 'F U T, 0, 0, 0',
	X =   -64.334  mm,	Y =   352.387  mm,	Z =     0.000  mm,
	W =  -167.363 deg,	P =     0.000 deg,	R =  -154.648 deg
};
P[854]{
   GP1:
	UF : 7, UT : 3,	CONFIG : 'F U T, 0, 0, 0',
	X =   -64.334  mm,	Y =   352.387  mm,	Z =     0.000  mm,
	W =  -167.363 deg,	P =     0.000 deg,	R =  -154.648 deg
};
P[855]{
   GP1:
	UF : 7, UT : 3,	CONFIG : 'F U T, 0, 0, 0',
	X =   -64.334  mm,	Y =   352.387  mm,	Z =     0.000  mm,
	W =  -167.363 deg,	P =     0.000 deg,	R =  -154.648 deg
};
P[856]{
   GP1:
	UF : 7, UT : 3,	CONFIG : 'F U T, 0, 0, 0',
	X =   -94.934  mm,	Y =   345.405  mm,	Z =     0.000  mm,
	W =  -167.364 deg,	P =     0.000 deg,	R =  -149.092 deg
};
P[857]{
   GP1:
	UF : 7, UT : 3,	CONFIG : 'F U T, 0, 0, 0',
	X =   -94.934  mm,	Y =   345.405  mm,	Z =     0.000  mm,
	W =  -167.364 deg,	P =     0.000 deg,	R =  -149.092 deg
};
P[858]{
   GP1:
	UF : 7, UT : 3,	CONFIG : 'F U T, 0, 0, 0',
	X =   -94.934  mm,	Y =   345.405  mm,	Z =     0.000  mm,
	W =  -167.364 deg,	P =     0.000 deg,	R =  -149.092 deg
};
P[859]{
   GP1:
	UF : 7, UT : 3,	CONFIG : 'F U T, 0, 0, 0',
	X =   -94.934  mm,	Y =   345.405  mm,	Z =     0.000  mm,
	W =  -167.364 deg,	P =     0.000 deg,	R =  -149.092 deg
};
P[860]{
   GP1:
	UF : 7, UT : 3,	CONFIG : 'F U T, 0, 0, 0',
	X =  -113.961  mm,	Y =   339.594  mm,	Z =     0.000  mm,
	W =  -167.365 deg,	P =     0.000 deg,	R =  -146.393 deg
};
P[861]{
   GP1:
	UF : 7, UT : 3,	CONFIG : 'F U T, 0, 0, 0',
	X =  -130.631  mm,	Y =   333.541  mm,	Z =     0.000  mm,
	W =  -167.366 deg,	P =     0.001 deg,	R =  -143.604 deg
};
P[862]{
   GP1:
	UF : 7, UT : 3,	CONFIG : 'F U T, 0, 0, 0',
	X =  -147.137  mm,	Y =   326.600  mm,	Z =     0.000  mm,
	W =  -167.367 deg,	P =     0.002 deg,	R =  -140.850 deg
};
P[863]{
   GP1:
	UF : 7, UT : 3,	CONFIG : 'F U T, 0, 0, 0',
	X =  -147.137  mm,	Y =   326.600  mm,	Z =     0.000  mm,
	W =  -167.367 deg,	P =     0.002 deg,	R =  -140.850 deg
};
P[864]{
   GP1:
	UF : 7, UT : 3,	CONFIG : 'F U T, 0, 0, 0',
	X =  -147.137  mm,	Y =   326.600  mm,	Z =     0.000  mm,
	W =  -167.367 deg,	P =     0.002 deg,	R =  -140.850 deg
};
P[865]{
   GP1:
	UF : 7, UT : 3,	CONFIG : 'F U T, 0, 0, 0',
	X =  -147.137  mm,	Y =   326.600  mm,	Z =     0.000  mm,
	W =  -167.367 deg,	P =     0.002 deg,	R =  -140.850 deg
};
P[866]{
   GP1:
	UF : 7, UT : 3,	CONFIG : 'F U T, 0, 0, 0',
	X =  -163.645  mm,	Y =   318.636  mm,	Z =     0.000  mm,
	W =  -167.370 deg,	P =     0.000 deg,	R =  -138.061 deg
};
P[867]{
   GP1:
	UF : 7, UT : 3,	CONFIG : 'F U T, 0, 0, 0',
	X =  -163.645  mm,	Y =   318.636  mm,	Z =     0.000  mm,
	W =  -167.370 deg,	P =     0.000 deg,	R =  -138.061 deg
};
P[868]{
   GP1:
	UF : 7, UT : 3,	CONFIG : 'F U T, 0, 0, 0',
	X =  -163.645  mm,	Y =   318.636  mm,	Z =     0.000  mm,
	W =  -167.370 deg,	P =     0.000 deg,	R =  -138.061 deg
};
P[869]{
   GP1:
	UF : 7, UT : 3,	CONFIG : 'F U T, 0, 0, 0',
	X =  -163.645  mm,	Y =   318.636  mm,	Z =     0.000  mm,
	W =  -167.370 deg,	P =     0.000 deg,	R =  -138.061 deg
};
P[870]{
   GP1:
	UF : 7, UT : 3,	CONFIG : 'F U T, 0, 0, 0',
	X =  -181.756  mm,	Y =   308.674  mm,	Z =     0.001  mm,
	W =  -167.368 deg,	P =    -0.004 deg,	R =  -134.437 deg
};
P[871]{
   GP1:
	UF : 7, UT : 3,	CONFIG : 'F U T, 0, 0, 0',
	X =  -200.158  mm,	Y =   297.075  mm,	Z =     0.006  mm,
	W =  -167.367 deg,	P =    -0.008 deg,	R =  -131.006 deg
};
P[872]{
   GP1:
	UF : 7, UT : 3,	CONFIG : 'F U T, 0, 0, 0',
	X =  -217.714  mm,	Y =   284.447  mm,	Z =     0.012  mm,
	W =  -167.367 deg,	P =    -0.012 deg,	R =  -127.556 deg
};
P[873]{
   GP1:
	UF : 7, UT : 3,	CONFIG : 'F U T, 0, 0, 0',
	X =  -234.191  mm,	Y =   271.054  mm,	Z =     0.020  mm,
	W =  -167.367 deg,	P =    -0.016 deg,	R =  -124.044 deg
};
P[874]{
   GP1:
	UF : 7, UT : 3,	CONFIG : 'F U T, 0, 0, 0',
	X =  -246.333  mm,	Y =   260.060  mm,	Z =     0.022  mm,
	W =  -167.388 deg,	P =     0.013 deg,	R =  -121.403 deg
};
P[875]{
   GP1:
	UF : 7, UT : 3,	CONFIG : 'F U T, 0, 0, 0',
	X =  -258.070  mm,	Y =   248.415  mm,	Z =     0.018  mm,
	W =  -167.406 deg,	P =     0.045 deg,	R =  -118.792 deg
};
P[876]{
   GP1:
	UF : 7, UT : 3,	CONFIG : 'F U T, 0, 0, 0',
	X =  -266.934  mm,	Y =   238.876  mm,	Z =     0.008  mm,
	W =  -167.463 deg,	P =     0.061 deg,	R =  -116.770 deg
};
P[877]{
   GP1:
	UF : 7, UT : 3,	CONFIG : 'F U T, 0, 0, 0',
	X =  -274.234  mm,	Y =   230.444  mm,	Z =     0.000  mm,
	W =  -167.509 deg,	P =     0.080 deg,	R =  -114.319 deg
};
P[878]{
   GP1:
	UF : 7, UT : 3,	CONFIG : 'F U T, 0, 0, 0',
	X =  -274.234  mm,	Y =   230.444  mm,	Z =     0.000  mm,
	W =  -167.509 deg,	P =     0.080 deg,	R =  -114.319 deg
};
P[879]{
   GP1:
	UF : 7, UT : 3,	CONFIG : 'F U T, 0, 0, 0',
	X =  -274.234  mm,	Y =   230.444  mm,	Z =     0.000  mm,
	W =  -167.509 deg,	P =     0.080 deg,	R =  -114.319 deg
};
P[880]{
   GP1:
	UF : 7, UT : 3,	CONFIG : 'F U T, 0, 0, 0',
	X =  -274.234  mm,	Y =   230.444  mm,	Z =     0.000  mm,
	W =  -167.509 deg,	P =     0.080 deg,	R =  -114.319 deg
};
P[881]{
   GP1:
	UF : 7, UT : 3,	CONFIG : 'F U T, 0, 0, 0',
	X =  -285.683  mm,	Y =   216.095  mm,	Z =     0.000  mm,
	W =  -167.656 deg,	P =     0.009 deg,	R =  -112.420 deg
};
P[882]{
   GP1:
	UF : 7, UT : 3,	CONFIG : 'F U T, 0, 0, 0',
	X =  -285.683  mm,	Y =   216.095  mm,	Z =     0.000  mm,
	W =  -167.656 deg,	P =     0.009 deg,	R =  -112.420 deg
};
P[883]{
   GP1:
	UF : 7, UT : 3,	CONFIG : 'F U T, 0, 0, 0',
	X =  -285.683  mm,	Y =   216.095  mm,	Z =     0.000  mm,
	W =  -167.656 deg,	P =     0.009 deg,	R =  -112.420 deg
};
P[884]{
   GP1:
	UF : 7, UT : 3,	CONFIG : 'F U T, 0, 0, 0',
	X =  -285.683  mm,	Y =   216.095  mm,	Z =     0.000  mm,
	W =  -167.656 deg,	P =     0.009 deg,	R =  -112.420 deg
};
P[885]{
   GP1:
	UF : 7, UT : 3,	CONFIG : 'F U T, 0, 0, 0',
	X =  -297.461  mm,	Y =   199.573  mm,	Z =     0.094  mm,
	W =  -167.858 deg,	P =    -0.457 deg,	R =  -108.720 deg
};
P[886]{
   GP1:
	UF : 7, UT : 3,	CONFIG : 'F U T, 0, 0, 0',
	X =  -306.395  mm,	Y =   185.562  mm,	Z =     0.395  mm,
	W =  -167.920 deg,	P =    -1.512 deg,	R =  -106.090 deg
};
P[887]{
   GP1:
	UF : 7, UT : 3,	CONFIG : 'F U T, 0, 0, 0',
	X =  -309.311  mm,	Y =   180.690  mm,	Z =     0.576  mm,
	W =  -167.907 deg,	P =    -1.920 deg,	R =  -105.231 deg
};
P[888]{
   GP1:
	UF : 7, UT : 3,	CONFIG : 'F U T, 0, 0, 0',
	X =  -313.246  mm,	Y =   173.778  mm,	Z =     0.866  mm,
	W =  -167.951 deg,	P =    -1.961 deg,	R =  -103.964 deg
};
P[889]{
   GP1:
	UF : 7, UT : 3,	CONFIG : 'F U T, 0, 0, 0',
	X =  -315.146  mm,	Y =   170.300  mm,	Z =     1.000  mm,
	W =  -167.986 deg,	P =    -1.720 deg,	R =  -103.253 deg
};
P[890]{
   GP1:
	UF : 7, UT : 3,	CONFIG : 'F U T, 0, 0, 0',
	X =  -315.146  mm,	Y =   170.300  mm,	Z =     1.000  mm,
	W =  -167.986 deg,	P =    -1.720 deg,	R =  -103.253 deg
};
P[891]{
   GP1:
	UF : 7, UT : 3,	CONFIG : 'F U T, 0, 0, 0',
	X =  -315.146  mm,	Y =   170.300  mm,	Z =     1.000  mm,
	W =  -167.986 deg,	P =    -1.720 deg,	R =  -103.253 deg
};
P[892]{
   GP1:
	UF : 7, UT : 3,	CONFIG : 'F U T, 0, 0, 0',
	X =  -315.146  mm,	Y =   170.300  mm,	Z =     1.000  mm,
	W =  -167.986 deg,	P =    -1.720 deg,	R =  -103.253 deg
};
P[893]{
   GP1:
	UF : 7, UT : 3,	CONFIG : 'F U T, 0, 0, 0',
	X =  -329.644  mm,	Y =   140.214  mm,	Z =     1.000  mm,
	W =  -167.177 deg,	P =     1.039 deg,	R =   -97.985 deg
};
P[894]{
   GP1:
	UF : 7, UT : 3,	CONFIG : 'F U T, 0, 0, 0',
	X =  -329.644  mm,	Y =   140.214  mm,	Z =     1.000  mm,
	W =  -167.177 deg,	P =     1.039 deg,	R =   -97.985 deg
};
P[895]{
   GP1:
	UF : 7, UT : 3,	CONFIG : 'F U T, 0, 0, 0',
	X =  -329.644  mm,	Y =   140.214  mm,	Z =     1.000  mm,
	W =  -167.177 deg,	P =     1.039 deg,	R =   -97.985 deg
};
P[896]{
   GP1:
	UF : 7, UT : 3,	CONFIG : 'F U T, 0, 0, 0',
	X =  -329.644  mm,	Y =   140.214  mm,	Z =     1.000  mm,
	W =  -167.177 deg,	P =     1.039 deg,	R =   -97.985 deg
};
P[897]{
   GP1:
	UF : 7, UT : 3,	CONFIG : 'F U T, 0, 0, 0',
	X =  -333.912  mm,	Y =   129.694  mm,	Z =     0.722  mm,
	W =  -167.179 deg,	P =     1.826 deg,	R =   -96.037 deg
};
P[898]{
   GP1:
	UF : 7, UT : 3,	CONFIG : 'F U T, 0, 0, 0',
	X =  -335.322  mm,	Y =   125.994  mm,	Z =     0.591  mm,
	W =  -167.288 deg,	P =     2.012 deg,	R =   -95.594 deg
};
P[899]{
   GP1:
	UF : 7, UT : 3,	CONFIG : 'F U T, 0, 0, 0',
	X =  -336.695  mm,	Y =   122.282  mm,	Z =     0.454  mm,
	W =  -167.411 deg,	P =     1.962 deg,	R =   -94.845 deg
};
P[900]{
   GP1:
	UF : 7, UT : 3,	CONFIG : 'F U T, 0, 0, 0',
	X =  -340.624  mm,	Y =   110.860  mm,	Z =     0.143  mm,
	W =  -167.673 deg,	P =     1.108 deg,	R =   -93.057 deg
};
P[901]{
   GP1:
	UF : 7, UT : 3,	CONFIG : 'F U T, 0, 0, 0',
	X =  -344.667  mm,	Y =    97.537  mm,	Z =     0.015  mm,
	W =  -167.578 deg,	P =     0.250 deg,	R =   -90.774 deg
};
P[902]{
   GP1:
	UF : 7, UT : 3,	CONFIG : 'F U T, 0, 0, 0',
	X =  -347.068  mm,	Y =    88.627  mm,	Z =     0.000  mm,
	W =  -167.508 deg,	P =     0.077 deg,	R =   -89.380 deg
};
P[903]{
   GP1:
	UF : 7, UT : 3,	CONFIG : 'F U T, 0, 0, 0',
	X =  -347.068  mm,	Y =    88.627  mm,	Z =     0.000  mm,
	W =  -167.508 deg,	P =     0.077 deg,	R =   -89.380 deg
};
P[904]{
   GP1:
	UF : 7, UT : 3,	CONFIG : 'F U T, 0, 0, 0',
	X =  -347.068  mm,	Y =    88.627  mm,	Z =     0.000  mm,
	W =  -167.508 deg,	P =     0.077 deg,	R =   -89.380 deg
};
P[905]{
   GP1:
	UF : 7, UT : 3,	CONFIG : 'F U T, 0, 0, 0',
	X =  -347.068  mm,	Y =    88.627  mm,	Z =     0.000  mm,
	W =  -167.508 deg,	P =     0.077 deg,	R =   -89.380 deg
};
P[906]{
   GP1:
	UF : 7, UT : 3,	CONFIG : 'F U T, 0, 0, 0',
	X =  -351.158  mm,	Y =    70.794  mm,	Z =     0.000  mm,
	W =  -167.419 deg,	P =     0.003 deg,	R =   -85.721 deg
};
P[907]{
   GP1:
	UF : 7, UT : 3,	CONFIG : 'F U T, 0, 0, 0',
	X =  -351.158  mm,	Y =    70.794  mm,	Z =     0.000  mm,
	W =  -167.419 deg,	P =     0.003 deg,	R =   -85.721 deg
};
P[908]{
   GP1:
	UF : 7, UT : 3,	CONFIG : 'F U T, 0, 0, 0',
	X =  -351.158  mm,	Y =    70.794  mm,	Z =     0.000  mm,
	W =  -167.419 deg,	P =     0.003 deg,	R =   -85.721 deg
};
P[909]{
   GP1:
	UF : 7, UT : 3,	CONFIG : 'F U T, 0, 0, 0',
	X =  -351.158  mm,	Y =    70.794  mm,	Z =     0.000  mm,
	W =  -167.419 deg,	P =     0.003 deg,	R =   -85.721 deg
};
P[910]{
   GP1:
	UF : 7, UT : 3,	CONFIG : 'F U T, 0, 1, 0',
	X =  -355.193  mm,	Y =    46.436  mm,	Z =     0.004  mm,
	W =  -167.399 deg,	P =     0.007 deg,	R =   -82.358 deg
};
P[911]{
   GP1:
	UF : 7, UT : 3,	CONFIG : 'F U T, 0, 1, 0',
	X =  -357.356  mm,	Y =    24.785  mm,	Z =     0.003  mm,
	W =  -167.381 deg,	P =     0.009 deg,	R =   -78.955 deg
};
P[912]{
   GP1:
	UF : 7, UT : 3,	CONFIG : 'F U T, 0, 1, 0',
	X =  -358.223  mm,	Y =     0.000  mm,	Z =     0.000  mm,
	W =  -167.361 deg,	P =     0.009 deg,	R =   -75.580 deg
};
P[913]{
   GP1:
	UF : 7, UT : 3,	CONFIG : 'F U T, 0, 1, 0',
	X =  -358.223  mm,	Y =     0.000  mm,	Z =     0.000  mm,
	W =  -167.361 deg,	P =     0.009 deg,	R =   -75.580 deg
};
P[914]{
   GP1:
	UF : 7, UT : 3,	CONFIG : 'F U T, 0, 1, 0',
	X =  -358.223  mm,	Y =     0.000  mm,	Z =     0.000  mm,
	W =  -167.361 deg,	P =     0.009 deg,	R =   -75.580 deg
};
P[915]{
   GP1:
	UF : 7, UT : 3,	CONFIG : 'F U T, 0, 1, 0',
	X =  -358.223  mm,	Y =     0.000  mm,	Z =     0.000  mm,
	W =  -167.361 deg,	P =     0.009 deg,	R =   -75.580 deg
};
P[916]{
   GP1:
	UF : 7, UT : 3,	CONFIG : 'F U T, 0, 1, 0',
	X =  -355.089  mm,	Y =     0.000  mm,	Z =     0.000  mm,
	W =  -167.361 deg,	P =     0.009 deg,	R =   -75.580 deg
};
P[917]{
   GP1:
	UF : 7, UT : 3,	CONFIG : 'F U T, 0, 1, 0',
	X =  -355.089  mm,	Y =     0.000  mm,	Z =     0.000  mm,
	W =  -167.361 deg,	P =     0.009 deg,	R =   -75.580 deg
};
P[918]{
   GP1:
	UF : 7, UT : 3,	CONFIG : 'F U T, 0, 1, 0',
	X =  -355.089  mm,	Y =     0.000  mm,	Z =     0.000  mm,
	W =  -167.361 deg,	P =     0.009 deg,	R =   -75.580 deg
};
P[919]{
   GP1:
	UF : 7, UT : 3,	CONFIG : 'F U T, 0, 1, 0',
	X =  -355.089  mm,	Y =     0.000  mm,	Z =     0.000  mm,
	W =  -167.361 deg,	P =     0.009 deg,	R =   -75.580 deg
};
P[920]{
   GP1:
	UF : 7, UT : 3,	CONFIG : 'F U T, 0, 1, 0',
	X =  -354.377  mm,	Y =    22.252  mm,	Z =     0.003  mm,
	W =  -167.375 deg,	P =     0.005 deg,	R =   -78.466 deg
};
P[921]{
   GP1:
	UF : 7, UT : 3,	CONFIG : 'F U T, 0, 1, 0',
	X =  -352.778  mm,	Y =    40.372  mm,	Z =     0.003  mm,
	W =  -167.386 deg,	P =     0.000 deg,	R =   -81.511 deg
};
P[922]{
   GP1:
	UF : 7, UT : 3,	CONFIG : 'F U T, 0, 1, 0',
	X =  -349.706  mm,	Y =    61.541  mm,	Z =     0.000  mm,
	W =  -167.399 deg,	P =    -0.007 deg,	R =   -84.454 deg
};
P[923]{
   GP1:
	UF : 7, UT : 3,	CONFIG : 'F U T, 0, 1, 0',
	X =  -349.706  mm,	Y =    61.541  mm,	Z =     0.000  mm,
	W =  -167.399 deg,	P =    -0.007 deg,	R =   -84.454 deg
};
P[924]{
   GP1:
	UF : 7, UT : 3,	CONFIG : 'F U T, 0, 1, 0',
	X =  -349.706  mm,	Y =    61.541  mm,	Z =     0.000  mm,
	W =  -167.399 deg,	P =    -0.007 deg,	R =   -84.454 deg
};
P[925]{
   GP1:
	UF : 7, UT : 3,	CONFIG : 'F U T, 0, 1, 0',
	X =  -349.706  mm,	Y =    61.541  mm,	Z =     0.000  mm,
	W =  -167.399 deg,	P =    -0.007 deg,	R =   -84.454 deg
};
P[926]{
   GP1:
	UF : 7, UT : 3,	CONFIG : 'F U T, 0, 0, 0',
	X =  -341.758  mm,	Y =    96.305  mm,	Z =     0.000  mm,
	W =  -167.575 deg,	P =     0.186 deg,	R =   -90.540 deg
};
P[927]{
   GP1:
	UF : 7, UT : 3,	CONFIG : 'F U T, 0, 0, 0',
	X =  -341.758  mm,	Y =    96.305  mm,	Z =     0.000  mm,
	W =  -167.575 deg,	P =     0.186 deg,	R =   -90.540 deg
};
P[928]{
   GP1:
	UF : 7, UT : 3,	CONFIG : 'F U T, 0, 0, 0',
	X =  -341.758  mm,	Y =    96.305  mm,	Z =     0.000  mm,
	W =  -167.575 deg,	P =     0.186 deg,	R =   -90.540 deg
};
P[929]{
   GP1:
	UF : 7, UT : 3,	CONFIG : 'F U T, 0, 0, 0',
	X =  -341.758  mm,	Y =    96.305  mm,	Z =     0.000  mm,
	W =  -167.575 deg,	P =     0.186 deg,	R =   -90.540 deg
};
P[930]{
   GP1:
	UF : 7, UT : 3,	CONFIG : 'F U T, 0, 0, 0',
	X =  -338.324  mm,	Y =   107.789  mm,	Z =     0.077  mm,
	W =  -167.700 deg,	P =     0.859 deg,	R =   -92.588 deg
};
P[931]{
   GP1:
	UF : 7, UT : 3,	CONFIG : 'F U T, 0, 0, 0',
	X =  -334.456  mm,	Y =   119.221  mm,	Z =     0.349  mm,
	W =  -167.582 deg,	P =     1.941 deg,	R =   -94.575 deg
};
P[932]{
   GP1:
	UF : 7, UT : 3,	CONFIG : 'F U T, 0, 0, 0',
	X =  -331.844  mm,	Y =   126.319  mm,	Z =     0.615  mm,
	W =  -167.403 deg,	P =     2.137 deg,	R =   -95.837 deg
};
P[933]{
   GP1:
	UF : 7, UT : 3,	CONFIG : 'F U T, 0, 0, 0',
	X =  -326.535  mm,	Y =   139.502  mm,	Z =     1.000  mm,
	W =  -167.386 deg,	P =     1.047 deg,	R =   -98.415 deg
};
P[934]{
   GP1:
	UF : 7, UT : 3,	CONFIG : 'F U T, 0, 0, 0',
	X =  -326.535  mm,	Y =   139.502  mm,	Z =     1.000  mm,
	W =  -167.386 deg,	P =     1.047 deg,	R =   -98.415 deg
};
P[935]{
   GP1:
	UF : 7, UT : 3,	CONFIG : 'F U T, 0, 0, 0',
	X =  -326.535  mm,	Y =   139.502  mm,	Z =     1.000  mm,
	W =  -167.386 deg,	P =     1.047 deg,	R =   -98.415 deg
};
P[936]{
   GP1:
	UF : 7, UT : 3,	CONFIG : 'F U T, 0, 0, 0',
	X =  -326.535  mm,	Y =   139.502  mm,	Z =     1.000  mm,
	W =  -167.386 deg,	P =     1.047 deg,	R =   -98.415 deg
};
P[937]{
   GP1:
	UF : 7, UT : 3,	CONFIG : 'F U T, 0, 0, 0',
	X =  -312.656  mm,	Y =   168.316  mm,	Z =     1.000  mm,
	W =  -168.257 deg,	P =    -1.511 deg,	R =  -103.413 deg
};
P[938]{
   GP1:
	UF : 7, UT : 3,	CONFIG : 'F U T, 0, 0, 0',
	X =  -312.656  mm,	Y =   168.316  mm,	Z =     1.000  mm,
	W =  -168.257 deg,	P =    -1.511 deg,	R =  -103.413 deg
};
P[939]{
   GP1:
	UF : 7, UT : 3,	CONFIG : 'F U T, 0, 0, 0',
	X =  -312.656  mm,	Y =   168.316  mm,	Z =     1.000  mm,
	W =  -168.257 deg,	P =    -1.511 deg,	R =  -103.413 deg
};
P[940]{
   GP1:
	UF : 7, UT : 3,	CONFIG : 'F U T, 0, 0, 0',
	X =  -312.656  mm,	Y =   168.316  mm,	Z =     1.000  mm,
	W =  -168.257 deg,	P =    -1.511 deg,	R =  -103.413 deg
};
P[941]{
   GP1:
	UF : 7, UT : 3,	CONFIG : 'F U T, 0, 0, 0',
	X =  -308.983  mm,	Y =   174.961  mm,	Z =     0.743  mm,
	W =  -168.162 deg,	P =    -1.948 deg,	R =  -104.573 deg
};
P[942]{
   GP1:
	UF : 7, UT : 3,	CONFIG : 'F U T, 0, 0, 0',
	X =  -304.968  mm,	Y =   181.863  mm,	Z =     0.458  mm,
	W =  -168.076 deg,	P =    -1.732 deg,	R =  -105.809 deg
};
P[943]{
   GP1:
	UF : 7, UT : 3,	CONFIG : 'F U T, 0, 0, 0',
	X =  -297.341  mm,	Y =   194.089  mm,	Z =     0.126  mm,
	W =  -167.975 deg,	P =    -0.683 deg,	R =  -108.148 deg
};
P[944]{
   GP1:
	UF : 7, UT : 3,	CONFIG : 'F U T, 0, 0, 0',
	X =  -288.373  mm,	Y =   207.174  mm,	Z =     0.000  mm,
	W =  -167.784 deg,	P =    -0.084 deg,	R =  -110.634 deg
};
P[945]{
   GP1:
	UF : 7, UT : 3,	CONFIG : 'F U T, 0, 0, 0',
	X =  -288.373  mm,	Y =   207.174  mm,	Z =     0.000  mm,
	W =  -167.784 deg,	P =    -0.084 deg,	R =  -110.634 deg
};
P[946]{
   GP1:
	UF : 7, UT : 3,	CONFIG : 'F U T, 0, 0, 0',
	X =  -288.373  mm,	Y =   207.174  mm,	Z =     0.000  mm,
	W =  -167.784 deg,	P =    -0.084 deg,	R =  -110.634 deg
};
P[947]{
   GP1:
	UF : 7, UT : 3,	CONFIG : 'F U T, 0, 0, 0',
	X =  -288.373  mm,	Y =   207.174  mm,	Z =     0.000  mm,
	W =  -167.784 deg,	P =    -0.084 deg,	R =  -110.634 deg
};
P[948]{
   GP1:
	UF : 7, UT : 3,	CONFIG : 'F U T, 0, 0, 0',
	X =  -266.135  mm,	Y =   235.048  mm,	Z =     0.000  mm,
	W =  -167.468 deg,	P =     0.094 deg,	R =  -115.890 deg
};
P[949]{
   GP1:
	UF : 7, UT : 3,	CONFIG : 'F U T, 0, 0, 0',
	X =  -266.135  mm,	Y =   235.048  mm,	Z =     0.000  mm,
	W =  -167.468 deg,	P =     0.094 deg,	R =  -115.890 deg
};
P[950]{
   GP1:
	UF : 7, UT : 3,	CONFIG : 'F U T, 0, 0, 0',
	X =  -266.135  mm,	Y =   235.048  mm,	Z =     0.000  mm,
	W =  -167.468 deg,	P =     0.094 deg,	R =  -115.890 deg
};
P[951]{
   GP1:
	UF : 7, UT : 3,	CONFIG : 'F U T, 0, 0, 0',
	X =  -266.135  mm,	Y =   235.048  mm,	Z =     0.000  mm,
	W =  -167.468 deg,	P =     0.094 deg,	R =  -115.890 deg
};
P[952]{
   GP1:
	UF : 7, UT : 3,	CONFIG : 'F U T, 0, 0, 0',
	X =  -254.396  mm,	Y =   247.717  mm,	Z =     0.016  mm,
	W =  -167.426 deg,	P =     0.046 deg,	R =  -119.162 deg
};
P[953]{
   GP1:
	UF : 7, UT : 3,	CONFIG : 'F U T, 0, 0, 0',
	X =  -241.307  mm,	Y =   260.480  mm,	Z =     0.022  mm,
	W =  -167.375 deg,	P =     0.002 deg,	R =  -122.176 deg
};
P[954]{
   GP1:
	UF : 7, UT : 3,	CONFIG : 'F U T, 0, 0, 0',
	X =  -224.340  mm,	Y =   275.231  mm,	Z =     0.016  mm,
	W =  -167.374 deg,	P =     0.001 deg,	R =  -125.792 deg
};
P[955]{
   GP1:
	UF : 7, UT : 3,	CONFIG : 'F U T, 0, 0, 0',
	X =  -206.491  mm,	Y =   288.871  mm,	Z =     0.008  mm,
	W =  -167.373 deg,	P =     0.000 deg,	R =  -129.371 deg
};
P[956]{
   GP1:
	UF : 7, UT : 3,	CONFIG : 'F U T, 0, 0, 0',
	X =  -187.758  mm,	Y =   301.372  mm,	Z =     0.003  mm,
	W =  -167.372 deg,	P =    -0.001 deg,	R =  -132.963 deg
};
P[957]{
   GP1:
	UF : 7, UT : 3,	CONFIG : 'F U T, 0, 0, 0',
	X =  -169.939  mm,	Y =   311.759  mm,	Z =     0.000  mm,
	W =  -167.371 deg,	P =    -0.002 deg,	R =  -136.930 deg
};
P[958]{
   GP1:
	UF : 7, UT : 3,	CONFIG : 'F U T, 0, 0, 0',
	X =  -169.939  mm,	Y =   311.759  mm,	Z =     0.000  mm,
	W =  -167.371 deg,	P =    -0.002 deg,	R =  -136.930 deg
};
P[959]{
   GP1:
	UF : 7, UT : 3,	CONFIG : 'F U T, 0, 0, 0',
	X =  -169.939  mm,	Y =   311.759  mm,	Z =     0.000  mm,
	W =  -167.371 deg,	P =    -0.002 deg,	R =  -136.930 deg
};
P[960]{
   GP1:
	UF : 7, UT : 3,	CONFIG : 'F U T, 0, 0, 0',
	X =  -169.939  mm,	Y =   311.759  mm,	Z =     0.000  mm,
	W =  -167.371 deg,	P =    -0.002 deg,	R =  -136.930 deg
};
P[961]{
   GP1:
	UF : 7, UT : 3,	CONFIG : 'F U T, 0, 0, 0',
	X =  -137.833  mm,	Y =   327.245  mm,	Z =     0.000  mm,
	W =  -167.366 deg,	P =     0.002 deg,	R =  -142.666 deg
};
P[962]{
   GP1:
	UF : 7, UT : 3,	CONFIG : 'F U T, 0, 0, 0',
	X =  -137.833  mm,	Y =   327.245  mm,	Z =     0.000  mm,
	W =  -167.366 deg,	P =     0.002 deg,	R =  -142.666 deg
};
P[963]{
   GP1:
	UF : 7, UT : 3,	CONFIG : 'F U T, 0, 0, 0',
	X =  -137.833  mm,	Y =   327.245  mm,	Z =     0.000  mm,
	W =  -167.366 deg,	P =     0.002 deg,	R =  -142.666 deg
};
P[964]{
   GP1:
	UF : 7, UT : 3,	CONFIG : 'F U T, 0, 0, 0',
	X =  -137.833  mm,	Y =   327.245  mm,	Z =     0.000  mm,
	W =  -167.366 deg,	P =     0.002 deg,	R =  -142.666 deg
};
P[965]{
   GP1:
	UF : 7, UT : 3,	CONFIG : 'F U T, 0, 0, 0',
	X =  -116.197  mm,	Y =   335.533  mm,	Z =     0.000  mm,
	W =  -167.365 deg,	P =     0.001 deg,	R =  -145.823 deg
};
P[966]{
   GP1:
	UF : 7, UT : 3,	CONFIG : 'F U T, 0, 0, 0',
	X =   -93.521  mm,	Y =   342.548  mm,	Z =     0.000  mm,
	W =  -167.363 deg,	P =     0.000 deg,	R =  -149.101 deg
};
P[967]{
   GP1:
	UF : 7, UT : 3,	CONFIG : 'F U T, 0, 0, 0',
	X =   -93.521  mm,	Y =   342.548  mm,	Z =     0.000  mm,
	W =  -167.363 deg,	P =     0.000 deg,	R =  -149.101 deg
};
P[968]{
   GP1:
	UF : 7, UT : 3,	CONFIG : 'F U T, 0, 0, 0',
	X =   -93.521  mm,	Y =   342.548  mm,	Z =     0.000  mm,
	W =  -167.363 deg,	P =     0.000 deg,	R =  -149.101 deg
};
P[969]{
   GP1:
	UF : 7, UT : 3,	CONFIG : 'F U T, 0, 0, 0',
	X =   -93.521  mm,	Y =   342.548  mm,	Z =     0.000  mm,
	W =  -167.363 deg,	P =     0.000 deg,	R =  -149.101 deg
};
P[970]{
   GP1:
	UF : 7, UT : 3,	CONFIG : 'F U T, 0, 0, 0',
	X =   -64.367  mm,	Y =   349.190  mm,	Z =     0.000  mm,
	W =  -167.363 deg,	P =     0.000 deg,	R =  -154.219 deg
};
P[971]{
   GP1:
	UF : 7, UT : 3,	CONFIG : 'F U T, 0, 0, 0',
	X =   -64.367  mm,	Y =   349.190  mm,	Z =     0.000  mm,
	W =  -167.363 deg,	P =     0.000 deg,	R =  -154.219 deg
};
P[972]{
   GP1:
	UF : 7, UT : 3,	CONFIG : 'F U T, 0, 0, 0',
	X =   -64.367  mm,	Y =   349.190  mm,	Z =     0.000  mm,
	W =  -167.363 deg,	P =     0.000 deg,	R =  -154.219 deg
};
P[973]{
   GP1:
	UF : 7, UT : 3,	CONFIG : 'F U T, 0, 0, 0',
	X =   -64.367  mm,	Y =   349.190  mm,	Z =     0.000  mm,
	W =  -167.363 deg,	P =     0.000 deg,	R =  -154.219 deg
};
P[974]{
   GP1:
	UF : 7, UT : 3,	CONFIG : 'F U T, 0, 0, 0',
	X =   -42.171  mm,	Y =   352.557  mm,	Z =     0.000  mm,
	W =  -167.363 deg,	P =     0.000 deg,	R =  -158.084 deg
};
P[975]{
   GP1:
	UF : 7, UT : 3,	CONFIG : 'F U T, 0, 0, 0',
	X =   -17.834  mm,	Y =   354.624  mm,	Z =     0.000  mm,
	W =  -167.364 deg,	P =     0.000 deg,	R =  -161.807 deg
};
P[976]{
   GP1:
	UF : 7, UT : 3,	CONFIG : 'F U T, 0, 0, 0',
	X =   -17.834  mm,	Y =   354.624  mm,	Z =     0.000  mm,
	W =  -167.364 deg,	P =     0.000 deg,	R =  -161.807 deg
};
P[977]{
   GP1:
	UF : 7, UT : 3,	CONFIG : 'F U T, 0, 0, 0',
	X =   -17.834  mm,	Y =   354.624  mm,	Z =     0.000  mm,
	W =  -167.364 deg,	P =     0.000 deg,	R =  -161.807 deg
};
P[978]{
   GP1:
	UF : 7, UT : 3,	CONFIG : 'F U T, 0, 0, 0',
	X =   -17.834  mm,	Y =   354.624  mm,	Z =     0.000  mm,
	W =  -167.364 deg,	P =     0.000 deg,	R =  -161.807 deg
};
P[979]{
   GP1:
	UF : 7, UT : 3,	CONFIG : 'F U T, 0, 0, 0',
	X =    17.834  mm,	Y =   354.624  mm,	Z =     0.000  mm,
	W =  -167.364 deg,	P =     0.000 deg,	R =  -168.087 deg
};
P[980]{
   GP1:
	UF : 7, UT : 3,	CONFIG : 'F U T, 0, 0, 0',
	X =    17.834  mm,	Y =   354.624  mm,	Z =     0.000  mm,
	W =  -167.364 deg,	P =     0.000 deg,	R =  -168.087 deg
};
P[981]{
   GP1:
	UF : 7, UT : 3,	CONFIG : 'F U T, 0, 0, 0',
	X =    17.834  mm,	Y =   354.624  mm,	Z =     0.000  mm,
	W =  -167.364 deg,	P =     0.000 deg,	R =  -168.087 deg
};
P[982]{
   GP1:
	UF : 7, UT : 3,	CONFIG : 'F U T, 0, 0, 0',
	X =    17.834  mm,	Y =   354.624  mm,	Z =     0.000  mm,
	W =  -167.364 deg,	P =     0.000 deg,	R =  -168.087 deg
};
P[983]{
   GP1:
	UF : 7, UT : 3,	CONFIG : 'F U T, 0, 0, 0',
	X =    42.148  mm,	Y =   352.560  mm,	Z =     0.000  mm,
	W =  -167.363 deg,	P =     0.000 deg,	R =  -171.819 deg
};
P[984]{
   GP1:
	UF : 7, UT : 3,	CONFIG : 'F U T, 0, 0, 0',
	X =    64.367  mm,	Y =   349.190  mm,	Z =     0.000  mm,
	W =  -167.363 deg,	P =     0.000 deg,	R =  -175.676 deg
};
P[985]{
   GP1:
	UF : 7, UT : 3,	CONFIG : 'F U T, 0, 0, 0',
	X =    64.367  mm,	Y =   349.190  mm,	Z =     0.000  mm,
	W =  -167.363 deg,	P =     0.000 deg,	R =  -175.676 deg
};
P[986]{
   GP1:
	UF : 7, UT : 3,	CONFIG : 'F U T, 0, 0, 0',
	X =    64.367  mm,	Y =   349.190  mm,	Z =     0.000  mm,
	W =  -167.363 deg,	P =     0.000 deg,	R =  -175.676 deg
};
P[987]{
   GP1:
	UF : 7, UT : 3,	CONFIG : 'F U T, 0, 0, 0',
	X =    64.367  mm,	Y =   349.190  mm,	Z =     0.000  mm,
	W =  -167.363 deg,	P =     0.000 deg,	R =  -175.676 deg
};
P[988]{
   GP1:
	UF : 7, UT : 3,	CONFIG : 'F U T, 0, 0, 0',
	X =    93.521  mm,	Y =   342.548  mm,	Z =     0.000  mm,
	W =  -167.363 deg,	P =     0.000 deg,	R =   179.208 deg
};
P[989]{
   GP1:
	UF : 7, UT : 3,	CONFIG : 'F U T, 0, 0, 0',
	X =    93.521  mm,	Y =   342.548  mm,	Z =     0.000  mm,
	W =  -167.363 deg,	P =     0.000 deg,	R =   179.208 deg
};
P[990]{
   GP1:
	UF : 7, UT : 3,	CONFIG : 'F U T, 0, 0, 0',
	X =    93.521  mm,	Y =   342.548  mm,	Z =     0.000  mm,
	W =  -167.363 deg,	P =     0.000 deg,	R =   179.208 deg
};
P[991]{
   GP1:
	UF : 7, UT : 3,	CONFIG : 'F U T, 0, 0, 0',
	X =    93.521  mm,	Y =   342.548  mm,	Z =     0.000  mm,
	W =  -167.363 deg,	P =     0.000 deg,	R =   179.208 deg
};
P[992]{
   GP1:
	UF : 7, UT : 3,	CONFIG : 'F U T, 0, 0, 0',
	X =   116.249  mm,	Y =   335.518  mm,	Z =     0.000  mm,
	W =  -167.364 deg,	P =     0.000 deg,	R =   175.919 deg
};
P[993]{
   GP1:
	UF : 7, UT : 3,	CONFIG : 'F U T, 0, 0, 0',
	X =   137.833  mm,	Y =   327.245  mm,	Z =     0.000  mm,
	W =  -167.364 deg,	P =     0.000 deg,	R =   172.775 deg
};
P[994]{
   GP1:
	UF : 7, UT : 3,	CONFIG : 'F U T, 0, 0, 0',
	X =   137.833  mm,	Y =   327.245  mm,	Z =     0.000  mm,
	W =  -167.364 deg,	P =     0.000 deg,	R =   172.775 deg
};
P[995]{
   GP1:
	UF : 7, UT : 3,	CONFIG : 'F U T, 0, 0, 0',
	X =   137.833  mm,	Y =   327.245  mm,	Z =     0.000  mm,
	W =  -167.364 deg,	P =     0.000 deg,	R =   172.775 deg
};
P[996]{
   GP1:
	UF : 7, UT : 3,	CONFIG : 'F U T, 0, 0, 0',
	X =   137.833  mm,	Y =   327.245  mm,	Z =     0.000  mm,
	W =  -167.364 deg,	P =     0.000 deg,	R =   172.775 deg
};
P[997]{
   GP1:
	UF : 7, UT : 3,	CONFIG : 'F U T, 0, 0, 0',
	X =   169.939  mm,	Y =   311.759  mm,	Z =     0.000  mm,
	W =  -167.364 deg,	P =     0.000 deg,	R =   167.036 deg
};
P[998]{
   GP1:
	UF : 7, UT : 3,	CONFIG : 'F U T, 0, 0, 0',
	X =   169.939  mm,	Y =   311.759  mm,	Z =     0.000  mm,
	W =  -167.364 deg,	P =     0.000 deg,	R =   167.036 deg
};
P[999]{
   GP1:
	UF : 7, UT : 3,	CONFIG : 'F U T, 0, 0, 0',
	X =   169.939  mm,	Y =   311.759  mm,	Z =     0.000  mm,
	W =  -167.364 deg,	P =     0.000 deg,	R =   167.036 deg
};
P[1000]{
   GP1:
	UF : 7, UT : 3,	CONFIG : 'F U T, 0, 0, 0',
	X =   169.939  mm,	Y =   311.759  mm,	Z =     0.000  mm,
	W =  -167.364 deg,	P =     0.000 deg,	R =   167.036 deg
};
P[1001]{
   GP1:
	UF : 7, UT : 3,	CONFIG : 'F U T, 0, 0, 0',
	X =   186.866  mm,	Y =   301.936  mm,	Z =     0.000  mm,
	W =  -167.364 deg,	P =     0.000 deg,	R =   163.269 deg
};
P[1002]{
   GP1:
	UF : 7, UT : 3,	CONFIG : 'F U T, 0, 0, 0',
	X =   204.856  mm,	Y =   290.021  mm,	Z =     0.000  mm,
	W =  -167.364 deg,	P =     0.000 deg,	R =   159.904 deg
};
P[1003]{
   GP1:
	UF : 7, UT : 3,	CONFIG : 'F U T, 0, 0, 0',
	X =   221.357  mm,	Y =   277.623  mm,	Z =     0.001  mm,
	W =  -167.364 deg,	P =     0.000 deg,	R =   156.434 deg
};
P[1004]{
   GP1:
	UF : 7, UT : 3,	CONFIG : 'F U T, 0, 0, 0',
	X =   237.471  mm,	Y =   263.983  mm,	Z =     0.000  mm,
	W =  -167.364 deg,	P =     0.000 deg,	R =   153.042 deg
};
P[1005]{
   GP1:
	UF : 7, UT : 3,	CONFIG : 'F U T, 0, 0, 0',
	X =   252.827  mm,	Y =   249.320  mm,	Z =     0.000  mm,
	W =  -167.365 deg,	P =     0.000 deg,	R =   149.686 deg
};
P[1006]{
   GP1:
	UF : 7, UT : 3,	CONFIG : 'F U T, 0, 0, 0',
	X =   266.135  mm,	Y =   235.048  mm,	Z =     0.000  mm,
	W =  -167.365 deg,	P =     0.000 deg,	R =   145.923 deg
};
P[1007]{
   GP1:
	UF : 7, UT : 3,	CONFIG : 'F U T, 0, 0, 0',
	X =   266.135  mm,	Y =   235.048  mm,	Z =     0.000  mm,
	W =  -167.365 deg,	P =     0.000 deg,	R =   145.923 deg
};
P[1008]{
   GP1:
	UF : 7, UT : 3,	CONFIG : 'F U T, 0, 0, 0',
	X =   266.135  mm,	Y =   235.048  mm,	Z =     0.000  mm,
	W =  -167.365 deg,	P =     0.000 deg,	R =   145.923 deg
};
P[1009]{
   GP1:
	UF : 7, UT : 3,	CONFIG : 'F U T, 0, 0, 0',
	X =   266.135  mm,	Y =   235.048  mm,	Z =     0.000  mm,
	W =  -167.365 deg,	P =     0.000 deg,	R =   145.923 deg
};
P[1010]{
   GP1:
	UF : 7, UT : 3,	CONFIG : 'F U T, 0, 0, 0',
	X =   288.373  mm,	Y =   207.174  mm,	Z =     0.000  mm,
	W =  -167.365 deg,	P =     0.001 deg,	R =   140.722 deg
};
P[1011]{
   GP1:
	UF : 7, UT : 3,	CONFIG : 'F U T, 0, 0, 0',
	X =   288.373  mm,	Y =   207.174  mm,	Z =     0.000  mm,
	W =  -167.365 deg,	P =     0.001 deg,	R =   140.722 deg
};
P[1012]{
   GP1:
	UF : 7, UT : 3,	CONFIG : 'F U T, 0, 0, 0',
	X =   288.373  mm,	Y =   207.174  mm,	Z =     0.000  mm,
	W =  -167.365 deg,	P =     0.001 deg,	R =   140.722 deg
};
P[1013]{
   GP1:
	UF : 7, UT : 3,	CONFIG : 'F U T, 0, 0, 0',
	X =   288.373  mm,	Y =   207.174  mm,	Z =     0.000  mm,
	W =  -167.365 deg,	P =     0.001 deg,	R =   140.722 deg
};
P[1014]{
   GP1:
	UF : 7, UT : 3,	CONFIG : 'F U T, 0, 0, 0',
	X =   301.002  mm,	Y =   188.350  mm,	Z =     0.000  mm,
	W =  -167.364 deg,	P =     0.000 deg,	R =   137.129 deg
};
P[1015]{
   GP1:
	UF : 7, UT : 3,	CONFIG : 'F U T, 0, 0, 0',
	X =   313.141  mm,	Y =   167.396  mm,	Z =     0.000  mm,
	W =  -167.363 deg,	P =     0.000 deg,	R =   133.557 deg
};
P[1016]{
   GP1:
	UF : 7, UT : 3,	CONFIG : 'F U T, 0, 0, 0',
	X =   313.141  mm,	Y =   167.396  mm,	Z =     0.000  mm,
	W =  -167.363 deg,	P =     0.000 deg,	R =   133.557 deg
};
P[1017]{
   GP1:
	UF : 7, UT : 3,	CONFIG : 'F U T, 0, 0, 0',
	X =   313.141  mm,	Y =   167.396  mm,	Z =     0.000  mm,
	W =  -167.363 deg,	P =     0.000 deg,	R =   133.557 deg
};
P[1018]{
   GP1:
	UF : 7, UT : 3,	CONFIG : 'F U T, 0, 0, 0',
	X =   313.141  mm,	Y =   167.396  mm,	Z =     0.000  mm,
	W =  -167.363 deg,	P =     0.000 deg,	R =   133.557 deg
};
P[1019]{
   GP1:
	UF : 7, UT : 3,	CONFIG : 'F U T, 0, 0, 0',
	X =   326.109  mm,	Y =   140.453  mm,	Z =     0.000  mm,
	W =  -167.363 deg,	P =     0.001 deg,	R =   128.873 deg
};
P[1020]{
   GP1:
	UF : 7, UT : 3,	CONFIG : 'F U T, 0, 0, 0',
	X =   326.109  mm,	Y =   140.453  mm,	Z =     0.000  mm,
	W =  -167.363 deg,	P =     0.001 deg,	R =   128.873 deg
};
P[1021]{
   GP1:
	UF : 7, UT : 3,	CONFIG : 'F U T, 0, 0, 0',
	X =   326.109  mm,	Y =   140.453  mm,	Z =     0.000  mm,
	W =  -167.363 deg,	P =     0.001 deg,	R =   128.873 deg
};
P[1022]{
   GP1:
	UF : 7, UT : 3,	CONFIG : 'F U T, 0, 0, 0',
	X =   326.109  mm,	Y =   140.453  mm,	Z =     0.000  mm,
	W =  -167.363 deg,	P =     0.001 deg,	R =   128.873 deg
};
P[1023]{
   GP1:
	UF : 7, UT : 3,	CONFIG : 'F U T, 0, 0, 0',
	X =   331.698  mm,	Y =   126.687  mm,	Z =     0.000  mm,
	W =  -167.364 deg,	P =     0.000 deg,	R =   125.956 deg
};
P[1024]{
   GP1:
	UF : 7, UT : 3,	CONFIG : 'F U T, 0, 0, 0',
	X =   337.232  mm,	Y =   111.128  mm,	Z =     0.000  mm,
	W =  -167.364 deg,	P =     0.000 deg,	R =   123.339 deg
};
P[1025]{
   GP1:
	UF : 7, UT : 3,	CONFIG : 'F U T, 0, 0, 0',
	X =   341.758  mm,	Y =    96.305  mm,	Z =     0.000  mm,
	W =  -167.365 deg,	P =     0.000 deg,	R =   120.625 deg
};
P[1026]{
   GP1:
	UF : 7, UT : 3,	CONFIG : 'F U T, 0, 0, 0',
	X =   341.758  mm,	Y =    96.305  mm,	Z =     0.000  mm,
	W =  -167.365 deg,	P =     0.000 deg,	R =   120.625 deg
};
P[1027]{
   GP1:
	UF : 7, UT : 3,	CONFIG : 'F U T, 0, 0, 0',
	X =   341.758  mm,	Y =    96.305  mm,	Z =     0.000  mm,
	W =  -167.365 deg,	P =     0.000 deg,	R =   120.625 deg
};
P[1028]{
   GP1:
	UF : 7, UT : 3,	CONFIG : 'F U T, 0, 0, 0',
	X =   341.758  mm,	Y =    96.305  mm,	Z =     0.000  mm,
	W =  -167.365 deg,	P =     0.000 deg,	R =   120.625 deg
};
P[1029]{
   GP1:
	UF : 7, UT : 3,	CONFIG : 'F U T, 0, 0, 0',
	X =   349.706  mm,	Y =    61.541  mm,	Z =     0.000  mm,
	W =  -167.364 deg,	P =     0.001 deg,	R =   114.560 deg
};
P[1030]{
   GP1:
	UF : 7, UT : 3,	CONFIG : 'F U T, 0, 0, 0',
	X =   349.706  mm,	Y =    61.541  mm,	Z =     0.000  mm,
	W =  -167.364 deg,	P =     0.001 deg,	R =   114.560 deg
};
P[1031]{
   GP1:
	UF : 7, UT : 3,	CONFIG : 'F U T, 0, 0, 0',
	X =   349.706  mm,	Y =    61.541  mm,	Z =     0.000  mm,
	W =  -167.364 deg,	P =     0.001 deg,	R =   114.560 deg
};
P[1032]{
   GP1:
	UF : 7, UT : 3,	CONFIG : 'F U T, 0, 0, 0',
	X =   349.706  mm,	Y =    61.541  mm,	Z =     0.000  mm,
	W =  -167.364 deg,	P =     0.001 deg,	R =   114.560 deg
};
P[1033]{
   GP1:
	UF : 7, UT : 3,	CONFIG : 'F U T, 0, 0, 0',
	X =   352.803  mm,	Y =    40.179  mm,	Z =     0.000  mm,
	W =  -167.364 deg,	P =     0.000 deg,	R =   111.598 deg
};
P[1034]{
   GP1:
	UF : 7, UT : 3,	CONFIG : 'F U T, 0, 0, 0',
	X =   354.386  mm,	Y =    22.086  mm,	Z =     0.000  mm,
	W =  -167.364 deg,	P =     0.000 deg,	R =   108.555 deg
};
P[1035]{
   GP1:
	UF : 7, UT : 3,	CONFIG : 'F U T, 0, 0, 0',
	X =   355.089  mm,	Y =     0.000  mm,	Z =     0.000  mm,
	W =  -167.364 deg,	P =    -0.001 deg,	R =   105.688 deg
};
P[1036]{
   GP1:
	UF : 7, UT : 3,	CONFIG : 'F U T, 0, 0, 0',
	X =   355.089  mm,	Y =     0.000  mm,	Z =     0.000  mm,
	W =  -167.364 deg,	P =    -0.001 deg,	R =   105.688 deg
};
P[1037]{
   GP1:
	UF : 7, UT : 3,	CONFIG : 'F U T, 0, 0, 0',
	X =   355.089  mm,	Y =     0.000  mm,	Z =     0.000  mm,
	W =  -167.364 deg,	P =    -0.001 deg,	R =   105.688 deg
};
P[1038]{
   GP1:
	UF : 7, UT : 3,	CONFIG : 'F U T, 0, 0, 0',
	X =   355.089  mm,	Y =     0.000  mm,	Z =     0.000  mm,
	W =  -167.364 deg,	P =    -0.001 deg,	R =   105.688 deg
};
P[1039]{
   GP1:
	UF : 7, UT : 3,	CONFIG : 'F U T, 0, 0, 0',
	X =   351.955  mm,	Y =     0.000  mm,	Z =     0.000  mm,
	W =  -167.364 deg,	P =    -0.001 deg,	R =   105.687 deg
};
P[1040]{
   GP1:
	UF : 7, UT : 3,	CONFIG : 'F U T, 0, 0, 0',
	X =   351.955  mm,	Y =     0.000  mm,	Z =     0.000  mm,
	W =  -167.364 deg,	P =    -0.001 deg,	R =   105.687 deg
};
P[1041]{
   GP1:
	UF : 7, UT : 3,	CONFIG : 'F U T, 0, 0, 0',
	X =   351.955  mm,	Y =     0.000  mm,	Z =     0.000  mm,
	W =  -167.364 deg,	P =    -0.001 deg,	R =   105.687 deg
};
P[1042]{
   GP1:
	UF : 7, UT : 3,	CONFIG : 'F U T, 0, 0, 0',
	X =   351.955  mm,	Y =     0.000  mm,	Z =     0.000  mm,
	W =  -167.364 deg,	P =    -0.001 deg,	R =   105.687 deg
};
P[1043]{
   GP1:
	UF : 7, UT : 3,	CONFIG : 'F U T, 0, 0, 0',
	X =   351.305  mm,	Y =    21.119  mm,	Z =     0.000  mm,
	W =  -167.364 deg,	P =     0.000 deg,	R =   108.463 deg
};
P[1044]{
   GP1:
	UF : 7, UT : 3,	CONFIG : 'F U T, 0, 0, 0',
	X =   349.822  mm,	Y =    38.574  mm,	Z =     0.000  mm,
	W =  -167.364 deg,	P =     0.000 deg,	R =   111.337 deg
};
P[1045]{
   GP1:
	UF : 7, UT : 3,	CONFIG : 'F U T, 0, 0, 0',
	X =   347.491  mm,	Y =    55.790  mm,	Z =     0.000  mm,
	W =  -167.364 deg,	P =     0.001 deg,	R =   114.212 deg
};
P[1046]{
   GP1:
	UF : 7, UT : 3,	CONFIG : 'F U T, 0, 0, 0',
	X =   347.491  mm,	Y =    55.790  mm,	Z =     0.000  mm,
	W =  -167.364 deg,	P =     0.001 deg,	R =   114.212 deg
};
P[1047]{
   GP1:
	UF : 7, UT : 3,	CONFIG : 'F U T, 0, 0, 0',
	X =   347.491  mm,	Y =    55.790  mm,	Z =     0.000  mm,
	W =  -167.364 deg,	P =     0.001 deg,	R =   114.212 deg
};
P[1048]{
   GP1:
	UF : 7, UT : 3,	CONFIG : 'F U T, 0, 0, 0',
	X =   347.491  mm,	Y =    55.790  mm,	Z =     0.000  mm,
	W =  -167.364 deg,	P =     0.001 deg,	R =   114.212 deg
};
P[1049]{
   GP1:
	UF : 7, UT : 3,	CONFIG : 'F U T, 0, 0, 0',
	X =   337.294  mm,	Y =   100.499  mm,	Z =     0.000  mm,
	W =  -167.365 deg,	P =    -0.001 deg,	R =   122.191 deg
};
P[1050]{
   GP1:
	UF : 7, UT : 3,	CONFIG : 'F U T, 0, 0, 0',
	X =   337.294  mm,	Y =   100.499  mm,	Z =     0.000  mm,
	W =  -167.365 deg,	P =    -0.001 deg,	R =   122.191 deg
};
P[1051]{
   GP1:
	UF : 7, UT : 3,	CONFIG : 'F U T, 0, 0, 0',
	X =   337.294  mm,	Y =   100.499  mm,	Z =     0.000  mm,
	W =  -167.365 deg,	P =    -0.001 deg,	R =   122.191 deg
};
P[1052]{
   GP1:
	UF : 7, UT : 3,	CONFIG : 'F U T, 0, 0, 0',
	X =   337.294  mm,	Y =   100.499  mm,	Z =     0.000  mm,
	W =  -167.365 deg,	P =    -0.001 deg,	R =   122.191 deg
};
P[1053]{
   GP1:
	UF : 7, UT : 3,	CONFIG : 'F U T, 0, 0, 0',
	X =   330.101  mm,	Y =   122.054  mm,	Z =     0.000  mm,
	W =  -167.364 deg,	P =     0.000 deg,	R =   125.352 deg
};
P[1054]{
   GP1:
	UF : 7, UT : 3,	CONFIG : 'F U T, 0, 0, 0',
	X =   322.696  mm,	Y =   140.444  mm,	Z =     0.000  mm,
	W =  -167.363 deg,	P =     0.001 deg,	R =   128.868 deg
};
P[1055]{
   GP1:
	UF : 7, UT : 3,	CONFIG : 'F U T, 0, 0, 0',
	X =   322.696  mm,	Y =   140.444  mm,	Z =     0.000  mm,
	W =  -167.363 deg,	P =     0.001 deg,	R =   128.868 deg
};
P[1056]{
   GP1:
	UF : 7, UT : 3,	CONFIG : 'F U T, 0, 0, 0',
	X =   322.696  mm,	Y =   140.444  mm,	Z =     0.000  mm,
	W =  -167.363 deg,	P =     0.001 deg,	R =   128.868 deg
};
P[1057]{
   GP1:
	UF : 7, UT : 3,	CONFIG : 'F U T, 0, 0, 0',
	X =   322.696  mm,	Y =   140.444  mm,	Z =     0.000  mm,
	W =  -167.363 deg,	P =     0.001 deg,	R =   128.868 deg
};
P[1058]{
   GP1:
	UF : 7, UT : 3,	CONFIG : 'F U T, 0, 0, 0',
	X =   311.016  mm,	Y =   164.743  mm,	Z =     0.000  mm,
	W =  -167.363 deg,	P =     0.000 deg,	R =   133.574 deg
};
P[1059]{
   GP1:
	UF : 7, UT : 3,	CONFIG : 'F U T, 0, 0, 0',
	X =   311.016  mm,	Y =   164.743  mm,	Z =     0.000  mm,
	W =  -167.363 deg,	P =     0.000 deg,	R =   133.574 deg
};
P[1060]{
   GP1:
	UF : 7, UT : 3,	CONFIG : 'F U T, 0, 0, 0',
	X =   311.016  mm,	Y =   164.743  mm,	Z =     0.000  mm,
	W =  -167.363 deg,	P =     0.000 deg,	R =   133.574 deg
};
P[1061]{
   GP1:
	UF : 7, UT : 3,	CONFIG : 'F U T, 0, 0, 0',
	X =   311.016  mm,	Y =   164.743  mm,	Z =     0.000  mm,
	W =  -167.363 deg,	P =     0.000 deg,	R =   133.574 deg
};
P[1062]{
   GP1:
	UF : 7, UT : 3,	CONFIG : 'F U T, 0, 0, 0',
	X =   299.331  mm,	Y =   185.111  mm,	Z =     0.000  mm,
	W =  -167.364 deg,	P =     0.000 deg,	R =   136.796 deg
};
P[1063]{
   GP1:
	UF : 7, UT : 3,	CONFIG : 'F U T, 0, 0, 0',
	X =   288.873  mm,	Y =   201.022  mm,	Z =     0.000  mm,
	W =  -167.364 deg,	P =     0.001 deg,	R =   140.270 deg
};
P[1064]{
   GP1:
	UF : 7, UT : 3,	CONFIG : 'F U T, 0, 0, 0',
	X =   288.873  mm,	Y =   201.022  mm,	Z =     0.000  mm,
	W =  -167.364 deg,	P =     0.001 deg,	R =   140.270 deg
};
P[1065]{
   GP1:
	UF : 7, UT : 3,	CONFIG : 'F U T, 0, 0, 0',
	X =   288.873  mm,	Y =   201.022  mm,	Z =     0.000  mm,
	W =  -167.364 deg,	P =     0.001 deg,	R =   140.270 deg
};
P[1066]{
   GP1:
	UF : 7, UT : 3,	CONFIG : 'F U T, 0, 0, 0',
	X =   288.873  mm,	Y =   201.022  mm,	Z =     0.000  mm,
	W =  -167.364 deg,	P =     0.001 deg,	R =   140.270 deg
};
P[1067]{
   GP1:
	UF : 7, UT : 3,	CONFIG : 'F U T, 0, 0, 0',
	X =   260.264  mm,	Y =   236.898  mm,	Z =     0.000  mm,
	W =  -167.365 deg,	P =     0.000 deg,	R =   147.278 deg
};
P[1068]{
   GP1:
	UF : 7, UT : 3,	CONFIG : 'F U T, 0, 0, 0',
	X =   260.264  mm,	Y =   236.898  mm,	Z =     0.000  mm,
	W =  -167.365 deg,	P =     0.000 deg,	R =   147.278 deg
};
P[1069]{
   GP1:
	UF : 7, UT : 3,	CONFIG : 'F U T, 0, 0, 0',
	X =   260.264  mm,	Y =   236.898  mm,	Z =     0.000  mm,
	W =  -167.365 deg,	P =     0.000 deg,	R =   147.278 deg
};
P[1070]{
   GP1:
	UF : 7, UT : 3,	CONFIG : 'F U T, 0, 0, 0',
	X =   260.264  mm,	Y =   236.898  mm,	Z =     0.000  mm,
	W =  -167.365 deg,	P =     0.000 deg,	R =   147.278 deg
};
P[1071]{
   GP1:
	UF : 7, UT : 3,	CONFIG : 'F U T, 0, 0, 0',
	X =   245.039  mm,	Y =   252.625  mm,	Z =     0.000  mm,
	W =  -167.365 deg,	P =     0.000 deg,	R =   150.981 deg
};
P[1072]{
   GP1:
	UF : 7, UT : 3,	CONFIG : 'F U T, 0, 0, 0',
	X =   228.476  mm,	Y =   267.700  mm,	Z =     0.001  mm,
	W =  -167.364 deg,	P =     0.000 deg,	R =   154.576 deg
};
P[1073]{
   GP1:
	UF : 7, UT : 3,	CONFIG : 'F U T, 0, 0, 0',
	X =   210.965  mm,	Y =   281.705  mm,	Z =     0.000  mm,
	W =  -167.364 deg,	P =     0.000 deg,	R =   158.213 deg
};
P[1074]{
   GP1:
	UF : 7, UT : 3,	CONFIG : 'F U T, 0, 0, 0',
	X =   192.764  mm,	Y =   294.457  mm,	Z =     0.000  mm,
	W =  -167.364 deg,	P =     0.000 deg,	R =   161.830 deg
};
P[1075]{
   GP1:
	UF : 7, UT : 3,	CONFIG : 'F U T, 0, 0, 0',
	X =   173.041  mm,	Y =   306.461  mm,	Z =     0.000  mm,
	W =  -167.364 deg,	P =     0.000 deg,	R =   165.373 deg
};
P[1076]{
   GP1:
	UF : 7, UT : 3,	CONFIG : 'F U T, 0, 0, 0',
	X =   173.041  mm,	Y =   306.461  mm,	Z =     0.000  mm,
	W =  -167.364 deg,	P =     0.000 deg,	R =   165.373 deg
};
P[1077]{
   GP1:
	UF : 7, UT : 3,	CONFIG : 'F U T, 0, 0, 0',
	X =   173.041  mm,	Y =   306.461  mm,	Z =     0.000  mm,
	W =  -167.364 deg,	P =     0.000 deg,	R =   165.373 deg
};
P[1078]{
   GP1:
	UF : 7, UT : 3,	CONFIG : 'F U T, 0, 0, 0',
	X =   173.041  mm,	Y =   306.461  mm,	Z =     0.000  mm,
	W =  -167.364 deg,	P =     0.000 deg,	R =   165.373 deg
};
P[1079]{
   GP1:
	UF : 7, UT : 3,	CONFIG : 'F U T, 0, 0, 0',
	X =   131.705  mm,	Y =   326.362  mm,	Z =     0.000  mm,
	W =  -167.364 deg,	P =     0.000 deg,	R =   172.497 deg
};
P[1080]{
   GP1:
	UF : 7, UT : 3,	CONFIG : 'F U T, 0, 0, 0',
	X =   131.705  mm,	Y =   326.362  mm,	Z =     0.000  mm,
	W =  -167.364 deg,	P =     0.000 deg,	R =   172.497 deg
};
P[1081]{
   GP1:
	UF : 7, UT : 3,	CONFIG : 'F U T, 0, 0, 0',
	X =   131.705  mm,	Y =   326.362  mm,	Z =     0.000  mm,
	W =  -167.364 deg,	P =     0.000 deg,	R =   172.497 deg
};
P[1082]{
   GP1:
	UF : 7, UT : 3,	CONFIG : 'F U T, 0, 0, 0',
	X =   131.705  mm,	Y =   326.362  mm,	Z =     0.000  mm,
	W =  -167.364 deg,	P =     0.000 deg,	R =   172.497 deg
};
P[1083]{
   GP1:
	UF : 7, UT : 3,	CONFIG : 'F U T, 0, 0, 0',
	X =   112.873  mm,	Y =   333.349  mm,	Z =     0.000  mm,
	W =  -167.364 deg,	P =     0.000 deg,	R =   176.402 deg
};
P[1084]{
   GP1:
	UF : 7, UT : 3,	CONFIG : 'F U T, 0, 0, 0',
	X =    91.398  mm,	Y =   339.871  mm,	Z =     0.000  mm,
	W =  -167.363 deg,	P =     0.000 deg,	R =   179.839 deg
};
P[1085]{
   GP1:
	UF : 7, UT : 3,	CONFIG : 'F U T, 0, 0, 0',
	X =    91.398  mm,	Y =   339.871  mm,	Z =     0.000  mm,
	W =  -167.363 deg,	P =     0.000 deg,	R =   179.839 deg
};
P[1086]{
   GP1:
	UF : 7, UT : 3,	CONFIG : 'F U T, 0, 0, 0',
	X =    91.398  mm,	Y =   339.871  mm,	Z =     0.000  mm,
	W =  -167.363 deg,	P =     0.000 deg,	R =   179.839 deg
};
P[1087]{
   GP1:
	UF : 7, UT : 3,	CONFIG : 'F U T, 0, 0, 0',
	X =    91.398  mm,	Y =   339.871  mm,	Z =     0.000  mm,
	W =  -167.363 deg,	P =     0.000 deg,	R =   179.839 deg
};
P[1088]{
   GP1:
	UF : 7, UT : 3,	CONFIG : 'F U T, 0, 0, 0',
	X =    65.113  mm,	Y =   345.858  mm,	Z =     0.000  mm,
	W =  -167.363 deg,	P =     0.000 deg,	R =  -176.396 deg
};
P[1089]{
   GP1:
	UF : 7, UT : 3,	CONFIG : 'F U T, 0, 0, 0',
	X =    65.113  mm,	Y =   345.858  mm,	Z =     0.000  mm,
	W =  -167.363 deg,	P =     0.000 deg,	R =  -176.396 deg
};
P[1090]{
   GP1:
	UF : 7, UT : 3,	CONFIG : 'F U T, 0, 0, 0',
	X =    65.113  mm,	Y =   345.858  mm,	Z =     0.000  mm,
	W =  -167.363 deg,	P =     0.000 deg,	R =  -176.396 deg
};
P[1091]{
   GP1:
	UF : 7, UT : 3,	CONFIG : 'F U T, 0, 0, 0',
	X =    65.113  mm,	Y =   345.858  mm,	Z =     0.000  mm,
	W =  -167.363 deg,	P =     0.000 deg,	R =  -176.396 deg
};
P[1092]{
   GP1:
	UF : 7, UT : 3,	CONFIG : 'F U T, 0, 0, 0',
	X =    45.890  mm,	Y =   348.940  mm,	Z =     0.000  mm,
	W =  -167.363 deg,	P =     0.000 deg,	R =  -172.413 deg
};
P[1093]{
   GP1:
	UF : 7, UT : 3,	CONFIG : 'F U T, 0, 0, 0',
	X =    22.921  mm,	Y =   351.203  mm,	Z =     0.000  mm,
	W =  -167.363 deg,	P =     0.000 deg,	R =  -169.115 deg
};
P[1094]{
   GP1:
	UF : 7, UT : 3,	CONFIG : 'F U T, 0, 0, 0',
	X =    22.921  mm,	Y =   351.203  mm,	Z =     0.000  mm,
	W =  -167.363 deg,	P =     0.000 deg,	R =  -169.115 deg
};
P[1095]{
   GP1:
	UF : 7, UT : 3,	CONFIG : 'F U T, 0, 0, 0',
	X =    22.921  mm,	Y =   351.203  mm,	Z =     0.000  mm,
	W =  -167.363 deg,	P =     0.000 deg,	R =  -169.115 deg
};
P[1096]{
   GP1:
	UF : 7, UT : 3,	CONFIG : 'F U T, 0, 0, 0',
	X =    22.921  mm,	Y =   351.203  mm,	Z =     0.000  mm,
	W =  -167.363 deg,	P =     0.000 deg,	R =  -169.115 deg
};
P[1097]{
   GP1:
	UF : 7, UT : 3,	CONFIG : 'F U T, 0, 0, 0',
	X =   -22.921  mm,	Y =   351.203  mm,	Z =     0.000  mm,
	W =  -167.364 deg,	P =     0.000 deg,	R =  -160.779 deg
};
P[1098]{
   GP1:
	UF : 7, UT : 3,	CONFIG : 'F U T, 0, 0, 0',
	X =   -22.921  mm,	Y =   351.203  mm,	Z =     0.000  mm,
	W =  -167.364 deg,	P =     0.000 deg,	R =  -160.779 deg
};
P[1099]{
   GP1:
	UF : 7, UT : 3,	CONFIG : 'F U T, 0, 0, 0',
	X =   -22.921  mm,	Y =   351.203  mm,	Z =     0.000  mm,
	W =  -167.364 deg,	P =     0.000 deg,	R =  -160.779 deg
};
P[1100]{
   GP1:
	UF : 7, UT : 3,	CONFIG : 'F U T, 0, 0, 0',
	X =   -22.921  mm,	Y =   351.203  mm,	Z =     0.000  mm,
	W =  -167.364 deg,	P =     0.000 deg,	R =  -160.779 deg
};
P[1101]{
   GP1:
	UF : 7, UT : 3,	CONFIG : 'F U T, 0, 0, 0',
	X =   -45.804  mm,	Y =   348.951  mm,	Z =     0.000  mm,
	W =  -167.363 deg,	P =     0.000 deg,	R =  -157.496 deg
};
P[1102]{
   GP1:
	UF : 7, UT : 3,	CONFIG : 'F U T, 0, 0, 0',
	X =   -65.113  mm,	Y =   345.858  mm,	Z =     0.000  mm,
	W =  -167.363 deg,	P =     0.000 deg,	R =  -153.619 deg
};
P[1103]{
   GP1:
	UF : 7, UT : 3,	CONFIG : 'F U T, 0, 0, 0',
	X =   -65.113  mm,	Y =   345.858  mm,	Z =     0.000  mm,
	W =  -167.363 deg,	P =     0.000 deg,	R =  -153.619 deg
};
P[1104]{
   GP1:
	UF : 7, UT : 3,	CONFIG : 'F U T, 0, 0, 0',
	X =   -65.113  mm,	Y =   345.858  mm,	Z =     0.000  mm,
	W =  -167.363 deg,	P =     0.000 deg,	R =  -153.619 deg
};
P[1105]{
   GP1:
	UF : 7, UT : 3,	CONFIG : 'F U T, 0, 0, 0',
	X =   -65.113  mm,	Y =   345.858  mm,	Z =     0.000  mm,
	W =  -167.363 deg,	P =     0.000 deg,	R =  -153.619 deg
};
P[1106]{
   GP1:
	UF : 7, UT : 3,	CONFIG : 'F U T, 0, 0, 0',
	X =   -91.398  mm,	Y =   339.871  mm,	Z =     0.000  mm,
	W =  -167.363 deg,	P =     0.000 deg,	R =  -149.714 deg
};
P[1107]{
   GP1:
	UF : 7, UT : 3,	CONFIG : 'F U T, 0, 0, 0',
	X =   -91.398  mm,	Y =   339.871  mm,	Z =     0.000  mm,
	W =  -167.363 deg,	P =     0.000 deg,	R =  -149.714 deg
};
P[1108]{
   GP1:
	UF : 7, UT : 3,	CONFIG : 'F U T, 0, 0, 0',
	X =   -91.398  mm,	Y =   339.871  mm,	Z =     0.000  mm,
	W =  -167.363 deg,	P =     0.000 deg,	R =  -149.714 deg
};
P[1109]{
   GP1:
	UF : 7, UT : 3,	CONFIG : 'F U T, 0, 0, 0',
	X =   -91.398  mm,	Y =   339.871  mm,	Z =     0.000  mm,
	W =  -167.363 deg,	P =     0.000 deg,	R =  -149.714 deg
};
P[1110]{
   GP1:
	UF : 7, UT : 3,	CONFIG : 'F U T, 0, 0, 0',
	X =  -112.866  mm,	Y =   333.353  mm,	Z =     0.000  mm,
	W =  -167.364 deg,	P =     0.001 deg,	R =  -146.314 deg
};
P[1111]{
   GP1:
	UF : 7, UT : 3,	CONFIG : 'F U T, 0, 0, 0',
	X =  -131.705  mm,	Y =   326.362  mm,	Z =     0.000  mm,
	W =  -167.365 deg,	P =     0.002 deg,	R =  -142.474 deg
};
P[1112]{
   GP1:
	UF : 7, UT : 3,	CONFIG : 'F U T, 0, 0, 0',
	X =  -131.705  mm,	Y =   326.362  mm,	Z =     0.000  mm,
	W =  -167.365 deg,	P =     0.002 deg,	R =  -142.474 deg
};
P[1113]{
   GP1:
	UF : 7, UT : 3,	CONFIG : 'F U T, 0, 0, 0',
	X =  -131.705  mm,	Y =   326.362  mm,	Z =     0.000  mm,
	W =  -167.365 deg,	P =     0.002 deg,	R =  -142.474 deg
};
P[1114]{
   GP1:
	UF : 7, UT : 3,	CONFIG : 'F U T, 0, 0, 0',
	X =  -131.705  mm,	Y =   326.362  mm,	Z =     0.000  mm,
	W =  -167.365 deg,	P =     0.002 deg,	R =  -142.474 deg
};
P[1115]{
   GP1:
	UF : 7, UT : 3,	CONFIG : 'F U T, 0, 0, 0',
	X =  -173.041  mm,	Y =   306.461  mm,	Z =     0.000  mm,
	W =  -167.372 deg,	P =    -0.003 deg,	R =  -135.227 deg
};
P[1116]{
   GP1:
	UF : 7, UT : 3,	CONFIG : 'F U T, 0, 0, 0',
	X =  -173.041  mm,	Y =   306.461  mm,	Z =     0.000  mm,
	W =  -167.372 deg,	P =    -0.003 deg,	R =  -135.227 deg
};
P[1117]{
   GP1:
	UF : 7, UT : 3,	CONFIG : 'F U T, 0, 0, 0',
	X =  -173.041  mm,	Y =   306.461  mm,	Z =     0.000  mm,
	W =  -167.372 deg,	P =    -0.003 deg,	R =  -135.227 deg
};
P[1118]{
   GP1:
	UF : 7, UT : 3,	CONFIG : 'F U T, 0, 0, 0',
	X =  -173.041  mm,	Y =   306.461  mm,	Z =     0.000  mm,
	W =  -167.372 deg,	P =    -0.003 deg,	R =  -135.227 deg
};
P[1119]{
   GP1:
	UF : 7, UT : 3,	CONFIG : 'F U T, 0, 0, 0',
	X =  -190.720  mm,	Y =   295.790  mm,	Z =     0.003  mm,
	W =  -167.372 deg,	P =    -0.002 deg,	R =  -132.163 deg
};
P[1120]{
   GP1:
	UF : 7, UT : 3,	CONFIG : 'F U T, 0, 0, 0',
	X =  -206.490  mm,	Y =   284.994  mm,	Z =     0.009  mm,
	W =  -167.373 deg,	P =    -0.002 deg,	R =  -128.960 deg
};
P[1121]{
   GP1:
	UF : 7, UT : 3,	CONFIG : 'F U T, 0, 0, 0',
	X =  -222.160  mm,	Y =   272.963  mm,	Z =     0.016  mm,
	W =  -167.373 deg,	P =    -0.001 deg,	R =  -125.844 deg
};
P[1122]{
   GP1:
	UF : 7, UT : 3,	CONFIG : 'F U T, 0, 0, 0',
	X =  -236.698  mm,	Y =   260.451  mm,	Z =     0.021  mm,
	W =  -167.374 deg,	P =     0.000 deg,	R =  -122.644 deg
};
P[1123]{
   GP1:
	UF : 7, UT : 3,	CONFIG : 'F U T, 0, 0, 0',
	X =  -249.147  mm,	Y =   248.563  mm,	Z =     0.016  mm,
	W =  -167.414 deg,	P =     0.050 deg,	R =  -119.969 deg
};
P[1124]{
   GP1:
	UF : 7, UT : 3,	CONFIG : 'F U T, 0, 0, 0',
	X =  -260.264  mm,	Y =   236.898  mm,	Z =     0.000  mm,
	W =  -167.447 deg,	P =     0.100 deg,	R =  -117.131 deg
};
P[1125]{
   GP1:
	UF : 7, UT : 3,	CONFIG : 'F U T, 0, 0, 0',
	X =  -260.264  mm,	Y =   236.898  mm,	Z =     0.000  mm,
	W =  -167.447 deg,	P =     0.100 deg,	R =  -117.131 deg
};
P[1126]{
   GP1:
	UF : 7, UT : 3,	CONFIG : 'F U T, 0, 0, 0',
	X =  -260.264  mm,	Y =   236.898  mm,	Z =     0.000  mm,
	W =  -167.447 deg,	P =     0.100 deg,	R =  -117.131 deg
};
P[1127]{
   GP1:
	UF : 7, UT : 3,	CONFIG : 'F U T, 0, 0, 0',
	X =  -260.264  mm,	Y =   236.898  mm,	Z =     0.000  mm,
	W =  -167.447 deg,	P =     0.100 deg,	R =  -117.131 deg
};
P[1128]{
   GP1:
	UF : 7, UT : 3,	CONFIG : 'F U T, 0, 0, 0',
	X =  -288.873  mm,	Y =   201.022  mm,	Z =     0.000  mm,
	W =  -167.893 deg,	P =    -0.197 deg,	R =  -110.313 deg
};
P[1129]{
   GP1:
	UF : 7, UT : 3,	CONFIG : 'F U T, 0, 0, 0',
	X =  -288.873  mm,	Y =   201.022  mm,	Z =     0.000  mm,
	W =  -167.893 deg,	P =    -0.197 deg,	R =  -110.313 deg
};
P[1130]{
   GP1:
	UF : 7, UT : 3,	CONFIG : 'F U T, 0, 0, 0',
	X =  -288.873  mm,	Y =   201.022  mm,	Z =     0.000  mm,
	W =  -167.893 deg,	P =    -0.197 deg,	R =  -110.313 deg
};
P[1131]{
   GP1:
	UF : 7, UT : 3,	CONFIG : 'F U T, 0, 0, 0',
	X =  -288.873  mm,	Y =   201.022  mm,	Z =     0.000  mm,
	W =  -167.893 deg,	P =    -0.197 deg,	R =  -110.313 deg
};
P[1132]{
   GP1:
	UF : 7, UT : 3,	CONFIG : 'F U T, 0, 0, 0',
	X =  -297.890  mm,	Y =   187.407  mm,	Z =     0.208  mm,
	W =  -168.125 deg,	P =    -1.096 deg,	R =  -107.109 deg
};
P[1133]{
   GP1:
	UF : 7, UT : 3,	CONFIG : 'F U T, 0, 0, 0',
	X =  -301.777  mm,	Y =   181.079  mm,	Z =     0.410  mm,
	W =  -168.208 deg,	P =    -1.678 deg,	R =  -106.017 deg
};
P[1134]{
   GP1:
	UF : 7, UT : 3,	CONFIG : 'F U T, 0, 0, 0',
	X =  -306.225  mm,	Y =   173.464  mm,	Z =     0.720  mm,
	W =  -168.359 deg,	P =    -1.852 deg,	R =  -104.630 deg
};
P[1135]{
   GP1:
	UF : 7, UT : 3,	CONFIG : 'F U T, 0, 0, 0',
	X =  -310.479  mm,	Y =   165.757  mm,	Z =     1.000  mm,
	W =  -168.472 deg,	P =    -1.237 deg,	R =  -103.508 deg
};
P[1136]{
   GP1:
	UF : 7, UT : 3,	CONFIG : 'F U T, 0, 0, 0',
	X =  -310.479  mm,	Y =   165.757  mm,	Z =     1.000  mm,
	W =  -168.472 deg,	P =    -1.237 deg,	R =  -103.508 deg
};
P[1137]{
   GP1:
	UF : 7, UT : 3,	CONFIG : 'F U T, 0, 0, 0',
	X =  -310.479  mm,	Y =   165.757  mm,	Z =     1.000  mm,
	W =  -168.472 deg,	P =    -1.237 deg,	R =  -103.508 deg
};
P[1138]{
   GP1:
	UF : 7, UT : 3,	CONFIG : 'F U T, 0, 0, 0',
	X =  -310.479  mm,	Y =   165.757  mm,	Z =     1.000  mm,
	W =  -168.472 deg,	P =    -1.237 deg,	R =  -103.508 deg
};
P[1139]{
   GP1:
	UF : 7, UT : 3,	CONFIG : 'F U T, 0, 0, 0',
	X =  -323.165  mm,	Y =   139.394  mm,	Z =     1.000  mm,
	W =  -167.595 deg,	P =     1.008 deg,	R =   -98.966 deg
};
P[1140]{
   GP1:
	UF : 7, UT : 3,	CONFIG : 'F U T, 0, 0, 0',
	X =  -323.165  mm,	Y =   139.394  mm,	Z =     1.000  mm,
	W =  -167.595 deg,	P =     1.008 deg,	R =   -98.966 deg
};
P[1141]{
   GP1:
	UF : 7, UT : 3,	CONFIG : 'F U T, 0, 0, 0',
	X =  -323.165  mm,	Y =   139.394  mm,	Z =     1.000  mm,
	W =  -167.595 deg,	P =     1.008 deg,	R =   -98.966 deg
};
P[1142]{
   GP1:
	UF : 7, UT : 3,	CONFIG : 'F U T, 0, 0, 0',
	X =  -323.165  mm,	Y =   139.394  mm,	Z =     1.000  mm,
	W =  -167.595 deg,	P =     1.008 deg,	R =   -98.966 deg
};
P[1143]{
   GP1:
	UF : 7, UT : 3,	CONFIG : 'F U T, 0, 0, 0',
	X =  -328.405  mm,	Y =   126.540  mm,	Z =     0.631  mm,
	W =  -167.514 deg,	P =     2.212 deg,	R =   -95.957 deg
};
P[1144]{
   GP1:
	UF : 7, UT : 3,	CONFIG : 'F U T, 0, 0, 0',
	X =  -330.738  mm,	Y =   120.311  mm,	Z =     0.385  mm,
	W =  -167.607 deg,	P =     2.141 deg,	R =   -94.815 deg
};
P[1145]{
   GP1:
	UF : 7, UT : 3,	CONFIG : 'F U T, 0, 0, 0',
	X =  -335.864  mm,	Y =   105.155  mm,	Z =     0.029  mm,
	W =  -167.677 deg,	P =     0.615 deg,	R =   -92.305 deg
};
P[1146]{
   GP1:
	UF : 7, UT : 3,	CONFIG : 'F U T, 0, 0, 0',
	X =  -337.294  mm,	Y =   100.499  mm,	Z =     0.000  mm,
	W =  -167.622 deg,	P =     0.306 deg,	R =   -92.059 deg
};
P[1147]{
   GP1:
	UF : 7, UT : 3,	CONFIG : 'F U T, 0, 0, 0',
	X =  -337.294  mm,	Y =   100.499  mm,	Z =     0.000  mm,
	W =  -167.622 deg,	P =     0.306 deg,	R =   -92.059 deg
};
P[1148]{
   GP1:
	UF : 7, UT : 3,	CONFIG : 'F U T, 0, 0, 0',
	X =  -337.294  mm,	Y =   100.499  mm,	Z =     0.000  mm,
	W =  -167.622 deg,	P =     0.306 deg,	R =   -92.059 deg
};
P[1149]{
   GP1:
	UF : 7, UT : 3,	CONFIG : 'F U T, 0, 0, 0',
	X =  -337.294  mm,	Y =   100.499  mm,	Z =     0.000  mm,
	W =  -167.622 deg,	P =     0.306 deg,	R =   -92.059 deg
};
P[1150]{
   GP1:
	UF : 7, UT : 3,	CONFIG : 'F U T, 0, 1, 0',
	X =  -347.491  mm,	Y =    55.790  mm,	Z =     0.000  mm,
	W =  -167.390 deg,	P =    -0.010 deg,	R =   -84.124 deg
};
P[1151]{
   GP1:
	UF : 7, UT : 3,	CONFIG : 'F U T, 0, 1, 0',
	X =  -347.491  mm,	Y =    55.790  mm,	Z =     0.000  mm,
	W =  -167.390 deg,	P =    -0.010 deg,	R =   -84.124 deg
};
P[1152]{
   GP1:
	UF : 7, UT : 3,	CONFIG : 'F U T, 0, 1, 0',
	X =  -347.491  mm,	Y =    55.790  mm,	Z =     0.000  mm,
	W =  -167.390 deg,	P =    -0.010 deg,	R =   -84.124 deg
};
P[1153]{
   GP1:
	UF : 7, UT : 3,	CONFIG : 'F U T, 0, 1, 0',
	X =  -347.491  mm,	Y =    55.790  mm,	Z =     0.000  mm,
	W =  -167.390 deg,	P =    -0.010 deg,	R =   -84.124 deg
};
P[1154]{
   GP1:
	UF : 7, UT : 3,	CONFIG : 'F U T, 0, 1, 0',
	X =  -349.820  mm,	Y =    38.586  mm,	Z =     0.003  mm,
	W =  -167.382 deg,	P =    -0.003 deg,	R =   -81.231 deg
};
P[1155]{
   GP1:
	UF : 7, UT : 3,	CONFIG : 'F U T, 0, 1, 0',
	X =  -351.303  mm,	Y =    21.167  mm,	Z =     0.003  mm,
	W =  -167.373 deg,	P =     0.003 deg,	R =   -78.345 deg
};
P[1156]{
   GP1:
	UF : 7, UT : 3,	CONFIG : 'F U T, 0, 1, 0',
	X =  -351.955  mm,	Y =     0.000  mm,	Z =     0.000  mm,
	W =  -167.361 deg,	P =     0.009 deg,	R =   -75.581 deg
};
P[1157]{
   GP1:
	UF : 7, UT : 3,	CONFIG : 'F U T, 0, 1, 0',
	X =  -351.955  mm,	Y =     0.000  mm,	Z =     0.000  mm,
	W =  -167.361 deg,	P =     0.009 deg,	R =   -75.581 deg
};
P[1158]{
   GP1:
	UF : 7, UT : 3,	CONFIG : 'F U T, 0, 1, 0',
	X =  -351.955  mm,	Y =     0.000  mm,	Z =     0.000  mm,
	W =  -167.361 deg,	P =     0.009 deg,	R =   -75.581 deg
};
P[1159]{
   GP1:
	UF : 7, UT : 3,	CONFIG : 'F U T, 0, 1, 0',
	X =  -351.955  mm,	Y =     0.000  mm,	Z =     0.000  mm,
	W =  -167.361 deg,	P =     0.009 deg,	R =   -75.581 deg
};
P[1160]{
   GP1:
	UF : 7, UT : 3,	CONFIG : 'F U T, 0, 1, 0',
	X =  -348.821  mm,	Y =     0.000  mm,	Z =     0.000  mm,
	W =  -167.361 deg,	P =     0.009 deg,	R =   -75.580 deg
};
P[1161]{
   GP1:
	UF : 7, UT : 3,	CONFIG : 'F U T, 0, 1, 0',
	X =  -348.821  mm,	Y =     0.000  mm,	Z =     0.000  mm,
	W =  -167.361 deg,	P =     0.009 deg,	R =   -75.580 deg
};
P[1162]{
   GP1:
	UF : 7, UT : 3,	CONFIG : 'F U T, 0, 1, 0',
	X =  -348.821  mm,	Y =     0.000  mm,	Z =     0.000  mm,
	W =  -167.361 deg,	P =     0.009 deg,	R =   -75.580 deg
};
P[1163]{
   GP1:
	UF : 7, UT : 3,	CONFIG : 'F U T, 0, 1, 0',
	X =  -348.821  mm,	Y =     0.000  mm,	Z =     0.000  mm,
	W =  -167.361 deg,	P =     0.009 deg,	R =   -75.580 deg
};
P[1164]{
   GP1:
	UF : 7, UT : 3,	CONFIG : 'F U T, 0, 1, 0',
	X =  -347.719  mm,	Y =    27.446  mm,	Z =     0.003  mm,
	W =  -167.374 deg,	P =    -0.001 deg,	R =   -79.422 deg
};
P[1165]{
   GP1:
	UF : 7, UT : 3,	CONFIG : 'F U T, 0, 1, 0',
	X =  -344.991  mm,	Y =    51.425  mm,	Z =     0.000  mm,
	W =  -167.384 deg,	P =    -0.011 deg,	R =   -83.308 deg
};
P[1166]{
   GP1:
	UF : 7, UT : 3,	CONFIG : 'F U T, 0, 1, 0',
	X =  -344.991  mm,	Y =    51.425  mm,	Z =     0.000  mm,
	W =  -167.384 deg,	P =    -0.011 deg,	R =   -83.308 deg
};
P[1167]{
   GP1:
	UF : 7, UT : 3,	CONFIG : 'F U T, 0, 1, 0',
	X =  -344.991  mm,	Y =    51.425  mm,	Z =     0.000  mm,
	W =  -167.384 deg,	P =    -0.011 deg,	R =   -83.308 deg
};
P[1168]{
   GP1:
	UF : 7, UT : 3,	CONFIG : 'F U T, 0, 1, 0',
	X =  -344.991  mm,	Y =    51.425  mm,	Z =     0.000  mm,
	W =  -167.384 deg,	P =    -0.011 deg,	R =   -83.308 deg
};
P[1169]{
   GP1:
	UF : 7, UT : 3,	CONFIG : 'F U T, 0, 0, 0',
	X =  -333.135  mm,	Y =   103.355  mm,	Z =     0.000  mm,
	W =  -167.638 deg,	P =     0.437 deg,	R =   -91.561 deg
};
P[1170]{
   GP1:
	UF : 7, UT : 3,	CONFIG : 'F U T, 0, 0, 0',
	X =  -333.135  mm,	Y =   103.355  mm,	Z =     0.000  mm,
	W =  -167.638 deg,	P =     0.437 deg,	R =   -91.561 deg
};
P[1171]{
   GP1:
	UF : 7, UT : 3,	CONFIG : 'F U T, 0, 0, 0',
	X =  -333.135  mm,	Y =   103.355  mm,	Z =     0.000  mm,
	W =  -167.638 deg,	P =     0.437 deg,	R =   -91.561 deg
};
P[1172]{
   GP1:
	UF : 7, UT : 3,	CONFIG : 'F U T, 0, 0, 0',
	X =  -333.135  mm,	Y =   103.355  mm,	Z =     0.000  mm,
	W =  -167.638 deg,	P =     0.437 deg,	R =   -91.561 deg
};
P[1173]{
   GP1:
	UF : 7, UT : 3,	CONFIG : 'F U T, 0, 0, 0',
	X =  -328.255  mm,	Y =   117.948  mm,	Z =     0.291  mm,
	W =  -167.684 deg,	P =     2.047 deg,	R =   -94.688 deg
};
P[1174]{
   GP1:
	UF : 7, UT : 3,	CONFIG : 'F U T, 0, 0, 0',
	X =  -325.878  mm,	Y =   124.367  mm,	Z =     0.545  mm,
	W =  -167.629 deg,	P =     2.346 deg,	R =   -95.800 deg
};
P[1175]{
   GP1:
	UF : 7, UT : 3,	CONFIG : 'F U T, 0, 0, 0',
	X =  -324.799  mm,	Y =   127.193  mm,	Z =     0.659  mm,
	W =  -167.621 deg,	P =     2.234 deg,	R =   -96.230 deg
};
P[1176]{
   GP1:
	UF : 7, UT : 3,	CONFIG : 'F U T, 0, 0, 0',
	X =  -319.450  mm,	Y =   140.081  mm,	Z =     1.000  mm,
	W =  -167.790 deg,	P =     0.910 deg,	R =   -98.471 deg
};
P[1177]{
   GP1:
	UF : 7, UT : 3,	CONFIG : 'F U T, 0, 0, 0',
	X =  -319.450  mm,	Y =   140.081  mm,	Z =     1.000  mm,
	W =  -167.790 deg,	P =     0.910 deg,	R =   -98.471 deg
};
P[1178]{
   GP1:
	UF : 7, UT : 3,	CONFIG : 'F U T, 0, 0, 0',
	X =  -319.450  mm,	Y =   140.081  mm,	Z =     1.000  mm,
	W =  -167.790 deg,	P =     0.910 deg,	R =   -98.471 deg
};
P[1179]{
   GP1:
	UF : 7, UT : 3,	CONFIG : 'F U T, 0, 0, 0',
	X =  -319.450  mm,	Y =   140.081  mm,	Z =     1.000  mm,
	W =  -167.790 deg,	P =     0.910 deg,	R =   -98.471 deg
};
P[1180]{
   GP1:
	UF : 7, UT : 3,	CONFIG : 'F U T, 0, 0, 0',
	X =  -308.698  mm,	Y =   162.429  mm,	Z =     1.000  mm,
	W =  -168.619 deg,	P =    -0.871 deg,	R =  -102.937 deg
};
P[1181]{
   GP1:
	UF : 7, UT : 3,	CONFIG : 'F U T, 0, 0, 0',
	X =  -308.698  mm,	Y =   162.429  mm,	Z =     1.000  mm,
	W =  -168.619 deg,	P =    -0.871 deg,	R =  -102.937 deg
};
P[1182]{
   GP1:
	UF : 7, UT : 3,	CONFIG : 'F U T, 0, 0, 0',
	X =  -308.698  mm,	Y =   162.429  mm,	Z =     1.000  mm,
	W =  -168.619 deg,	P =    -0.871 deg,	R =  -102.937 deg
};
P[1183]{
   GP1:
	UF : 7, UT : 3,	CONFIG : 'F U T, 0, 0, 0',
	X =  -308.698  mm,	Y =   162.429  mm,	Z =     1.000  mm,
	W =  -168.619 deg,	P =    -0.871 deg,	R =  -102.937 deg
};
P[1184]{
   GP1:
	UF : 7, UT : 3,	CONFIG : 'F U T, 0, 0, 0',
	X =  -304.278  mm,	Y =   170.562  mm,	Z =     0.741  mm,
	W =  -168.545 deg,	P =    -1.673 deg,	R =  -104.288 deg
};
P[1185]{
   GP1:
	UF : 7, UT : 3,	CONFIG : 'F U T, 0, 0, 0',
	X =  -299.991  mm,	Y =   177.979  mm,	Z =     0.443  mm,
	W =  -168.362 deg,	P =    -1.726 deg,	R =  -105.695 deg
};
P[1186]{
   GP1:
	UF : 7, UT : 3,	CONFIG : 'F U T, 0, 0, 0',
	X =  -288.517  mm,	Y =   196.042  mm,	Z =     0.000  mm,
	W =  -167.992 deg,	P =    -0.314 deg,	R =  -108.539 deg
};
P[1187]{
   GP1:
	UF : 7, UT : 3,	CONFIG : 'F U T, 0, 0, 0',
	X =  -288.517  mm,	Y =   196.042  mm,	Z =     0.000  mm,
	W =  -167.992 deg,	P =    -0.314 deg,	R =  -108.539 deg
};
P[1188]{
   GP1:
	UF : 7, UT : 3,	CONFIG : 'F U T, 0, 0, 0',
	X =  -288.517  mm,	Y =   196.042  mm,	Z =     0.000  mm,
	W =  -167.992 deg,	P =    -0.314 deg,	R =  -108.539 deg
};
P[1189]{
   GP1:
	UF : 7, UT : 3,	CONFIG : 'F U T, 0, 0, 0',
	X =  -288.517  mm,	Y =   196.042  mm,	Z =     0.000  mm,
	W =  -167.992 deg,	P =    -0.314 deg,	R =  -108.539 deg
};
P[1190]{
   GP1:
	UF : 7, UT : 3,	CONFIG : 'F U T, 0, 0, 0',
	X =  -255.318  mm,	Y =   237.661  mm,	Z =     0.000  mm,
	W =  -167.431 deg,	P =     0.104 deg,	R =  -118.108 deg
};
P[1191]{
   GP1:
	UF : 7, UT : 3,	CONFIG : 'F U T, 0, 0, 0',
	X =  -255.318  mm,	Y =   237.661  mm,	Z =     0.000  mm,
	W =  -167.431 deg,	P =     0.104 deg,	R =  -118.108 deg
};
P[1192]{
   GP1:
	UF : 7, UT : 3,	CONFIG : 'F U T, 0, 0, 0',
	X =  -255.318  mm,	Y =   237.661  mm,	Z =     0.000  mm,
	W =  -167.431 deg,	P =     0.104 deg,	R =  -118.108 deg
};
P[1193]{
   GP1:
	UF : 7, UT : 3,	CONFIG : 'F U T, 0, 0, 0',
	X =  -255.318  mm,	Y =   237.661  mm,	Z =     0.000  mm,
	W =  -167.431 deg,	P =     0.104 deg,	R =  -118.108 deg
};
P[1194]{
   GP1:
	UF : 7, UT : 3,	CONFIG : 'F U T, 0, 0, 0',
	X =  -244.166  mm,	Y =   249.102  mm,	Z =     0.017  mm,
	W =  -167.403 deg,	P =     0.049 deg,	R =  -120.505 deg
};
P[1195]{
   GP1:
	UF : 7, UT : 3,	CONFIG : 'F U T, 0, 0, 0',
	X =  -232.964  mm,	Y =   259.606  mm,	Z =     0.020  mm,
	W =  -167.373 deg,	P =    -0.001 deg,	R =  -123.022 deg
};
P[1196]{
   GP1:
	UF : 7, UT : 3,	CONFIG : 'F U T, 0, 0, 0',
	X =  -219.177  mm,	Y =   271.343  mm,	Z =     0.016  mm,
	W =  -167.373 deg,	P =    -0.002 deg,	R =  -126.041 deg
};
P[1197]{
   GP1:
	UF : 7, UT : 3,	CONFIG : 'F U T, 0, 0, 0',
	X =  -204.531  mm,	Y =   282.545  mm,	Z =     0.009  mm,
	W =  -167.373 deg,	P =    -0.003 deg,	R =  -129.005 deg
};
P[1198]{
   GP1:
	UF : 7, UT : 3,	CONFIG : 'F U T, 0, 0, 0',
	X =  -189.632  mm,	Y =   292.762  mm,	Z =     0.003  mm,
	W =  -167.373 deg,	P =    -0.004 deg,	R =  -132.024 deg
};
P[1199]{
   GP1:
	UF : 7, UT : 3,	CONFIG : 'F U T, 0, 0, 0',
	X =  -174.892  mm,	Y =   301.790  mm,	Z =     0.000  mm,
	W =  -167.372 deg,	P =    -0.005 deg,	R =  -135.243 deg
};
P[1200]{
   GP1:
	UF : 7, UT : 3,	CONFIG : 'F U T, 0, 0, 0',
	X =  -174.892  mm,	Y =   301.790  mm,	Z =     0.000  mm,
	W =  -167.372 deg,	P =    -0.005 deg,	R =  -135.243 deg
};
P[1201]{
   GP1:
	UF : 7, UT : 3,	CONFIG : 'F U T, 0, 0, 0',
	X =  -174.892  mm,	Y =   301.790  mm,	Z =     0.000  mm,
	W =  -167.372 deg,	P =    -0.005 deg,	R =  -135.243 deg
};
P[1202]{
   GP1:
	UF : 7, UT : 3,	CONFIG : 'F U T, 0, 0, 0',
	X =  -174.892  mm,	Y =   301.790  mm,	Z =     0.000  mm,
	W =  -167.372 deg,	P =    -0.005 deg,	R =  -135.243 deg
};
P[1203]{
   GP1:
	UF : 7, UT : 3,	CONFIG : 'F U T, 0, 0, 0',
	X =  -126.912  mm,	Y =   324.901  mm,	Z =     0.000  mm,
	W =  -167.365 deg,	P =     0.002 deg,	R =  -144.020 deg
};
P[1204]{
   GP1:
	UF : 7, UT : 3,	CONFIG : 'F U T, 0, 0, 0',
	X =  -126.912  mm,	Y =   324.901  mm,	Z =     0.000  mm,
	W =  -167.365 deg,	P =     0.002 deg,	R =  -144.020 deg
};
P[1205]{
   GP1:
	UF : 7, UT : 3,	CONFIG : 'F U T, 0, 0, 0',
	X =  -126.912  mm,	Y =   324.901  mm,	Z =     0.000  mm,
	W =  -167.365 deg,	P =     0.002 deg,	R =  -144.020 deg
};
P[1206]{
   GP1:
	UF : 7, UT : 3,	CONFIG : 'F U T, 0, 0, 0',
	X =  -126.912  mm,	Y =   324.901  mm,	Z =     0.000  mm,
	W =  -167.365 deg,	P =     0.002 deg,	R =  -144.020 deg
};
P[1207]{
   GP1:
	UF : 7, UT : 3,	CONFIG : 'F U T, 0, 0, 0',
	X =  -106.083  mm,	Y =   332.287  mm,	Z =     0.000  mm,
	W =  -167.364 deg,	P =     0.001 deg,	R =  -147.250 deg
};
P[1208]{
   GP1:
	UF : 7, UT : 3,	CONFIG : 'F U T, 0, 0, 0',
	X =   -88.319  mm,	Y =   337.433  mm,	Z =     0.000  mm,
	W =  -167.363 deg,	P =     0.000 deg,	R =  -150.913 deg
};
P[1209]{
   GP1:
	UF : 7, UT : 3,	CONFIG : 'F U T, 0, 0, 0',
	X =   -88.319  mm,	Y =   337.433  mm,	Z =     0.000  mm,
	W =  -167.363 deg,	P =     0.000 deg,	R =  -150.913 deg
};
P[1210]{
   GP1:
	UF : 7, UT : 3,	CONFIG : 'F U T, 0, 0, 0',
	X =   -88.319  mm,	Y =   337.433  mm,	Z =     0.000  mm,
	W =  -167.363 deg,	P =     0.000 deg,	R =  -150.913 deg
};
P[1211]{
   GP1:
	UF : 7, UT : 3,	CONFIG : 'F U T, 0, 0, 0',
	X =   -88.319  mm,	Y =   337.433  mm,	Z =     0.000  mm,
	W =  -167.363 deg,	P =     0.000 deg,	R =  -150.913 deg
};
P[1212]{
   GP1:
	UF : 7, UT : 3,	CONFIG : 'F U T, 0, 0, 0',
	X =   -66.816  mm,	Y =   342.344  mm,	Z =     0.000  mm,
	W =  -167.363 deg,	P =     0.000 deg,	R =  -154.099 deg
};
P[1213]{
   GP1:
